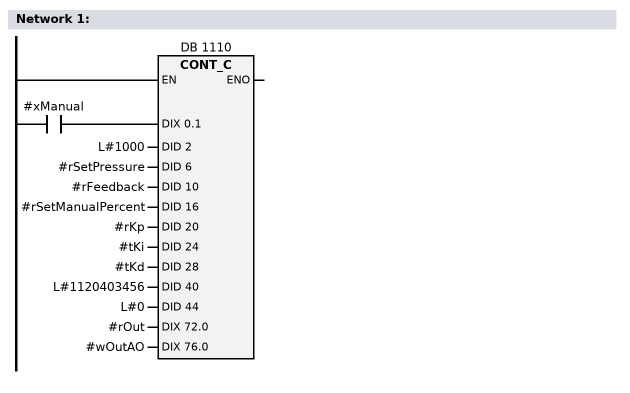
NETWORK
TITLE =
      A     #xManual;
      =     L 0.1;
      BLD   103;
      CALL  "CONT_C" , DB 1110 (
           DIX 0.1                  := L 0.1,
           DID 2                    := L#1000,
           DID 6                    := #rSetPressure,
           DID 10                   := #rFeedback,
           DID 16                   := #rSetManualPercent,
           DID 20                   := #rKp,
           DID 24                   := #tKi,
           DID 28                   := #tKd,
           DID 40                   := L#1120403456,
           DID 44                   := L#0,
           DIX 72.0                 := #rOut,
           DIX 76.0                 := #wOutAO);
      NOP   0;
END_FUNCTION_BLOCK

FUNCTION_BLOCK "fbPID"	// FB 34
VERSION : 0.1
BEGIN
// (block stored without names or comments; labels and parameter names are numbered)
END_FUNCTION_BLOCK

// FB 35: know-how protected block, not included

FUNCTION_BLOCK "DERIVATIVE"	// FB 36
VERSION : 0.0
VAR_INPUT
  IN : REAL ;
  TM : INT ;
  RESET : BOOL ;
END_VAR
VAR_OUTPUT
  OUT : REAL ;
END_VAR
VAR
  X3 : REAL ;
  X2 : REAL ;
  X1 : REAL ;
  T_2 : INT ;
  T_1 : INT ;
  INIT : BOOL  := TRUE;
END_VAR
BEGIN
// body was compiled from an SCL source; compiled code not shown
END_FUNCTION_BLOCK

FUNCTION_BLOCK "INTEGRAL"	// FB 37
VERSION : 0.0
VAR_INPUT
  IN : REAL ;
  TM : INT ;
  RESET : BOOL ;
END_VAR
VAR_OUTPUT
  OUT : REAL ;
  OVERFLOW : BOOL ;
END_VAR
BEGIN
// body was compiled from an SCL source; compiled code not shown
END_FUNCTION_BLOCK

FUNCTION_BLOCK "DO_Valve"	// FB 38
VERSION : 0.0
VAR_INPUT
  xCmdStop : BOOL ;
  xSnsOpn : BOOL ;
  xSnsCls : BOOL ;
  xAlm : BOOL ;
END_VAR
VAR_OUTPUT
  xDO_Opn : BOOL ;
  xDO_Cls : BOOL ;
  xDO_Stop : BOOL ;
END_VAR
VAR_IN_OUT
  xCmdOpn : BOOL ;
  xCmdCls : BOOL ;
END_VAR
VAR
  rtOn : BOOL ;
  rtOff : BOOL ;
  ftOn : BOOL ;
  ftOff : BOOL ;
  OpnOld : BOOL ;
  ClsOld : BOOL ;
END_VAR
BEGIN
// body was compiled from an SCL source; compiled code not shown
END_FUNCTION_BLOCK

FUNCTION_BLOCK "ValvesPrg"	// FB 39
VERSION : 0.1
BEGIN
NETWORK
TITLE =
NETWORK
TITLE =
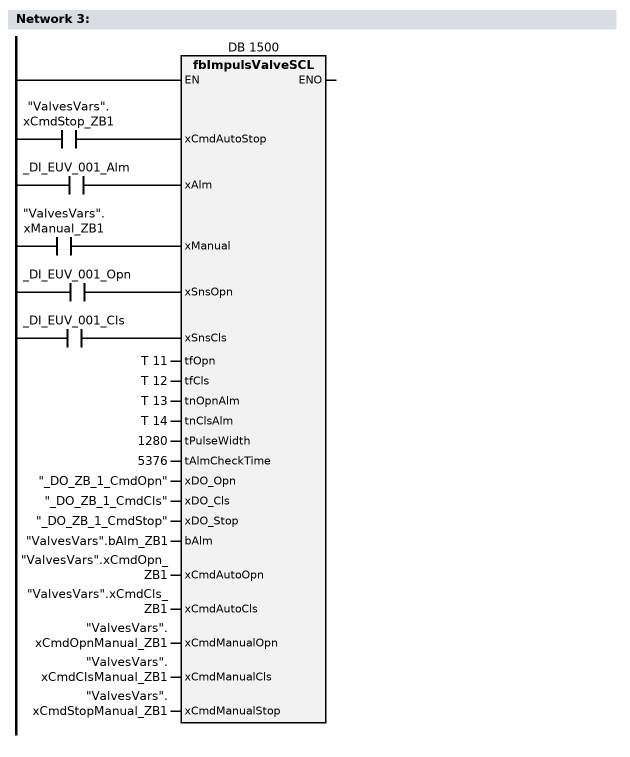
NETWORK
TITLE =
      A     "ValvesVars".xCmdStop_ZB1;
      =     L 0.0;
      BLD   103;
      A     "_DI_EUV_001_Alm";
      =     L 0.1;
      BLD   103;
      A     "ValvesVars".xManual_ZB1;
      =     L 0.2;
      BLD   103;
      A     "_DI_EUV_001_Opn";
      =     L 0.3;
      BLD   103;
      A     "_DI_EUV_001_Cls";
      =     L 0.4;
      BLD   103;
      CALL  "fbImpulsValveSCL" , DB 1500 (
           xCmdAutoStop             := L 0.0,
           xAlm                     := L 0.1,
           xManual                  := L 0.2,
           xSnsOpn                  := L 0.3,
           xSnsCls                  := L 0.4,
           tfOpn                    := T 11,
           tfCls                    := T 12,
           tnOpnAlm                 := T 13,
           tnClsAlm                 := T 14,
           tPulseWidth              := 1280,
           tAlmCheckTime            := 5376,
           xDO_Opn                  := "_DO_ZB_1_CmdOpn",
           xDO_Cls                  := "_DO_ZB_1_CmdCls",
           xDO_Stop                 := "_DO_ZB_1_CmdStop",
           bAlm                     := "ValvesVars".bAlm_ZB1,
           xCmdAutoOpn              := "ValvesVars".xCmdOpn_ZB1,
           xCmdAutoCls              := "ValvesVars".xCmdCls_ZB1,
           xCmdManualOpn            := "ValvesVars".xCmdOpnManual_ZB1,
           xCmdManualCls            := "ValvesVars".xCmdClsManual_ZB1,
           xCmdManualStop           := "ValvesVars".xCmdStopManual_ZB1);
      NOP   0;
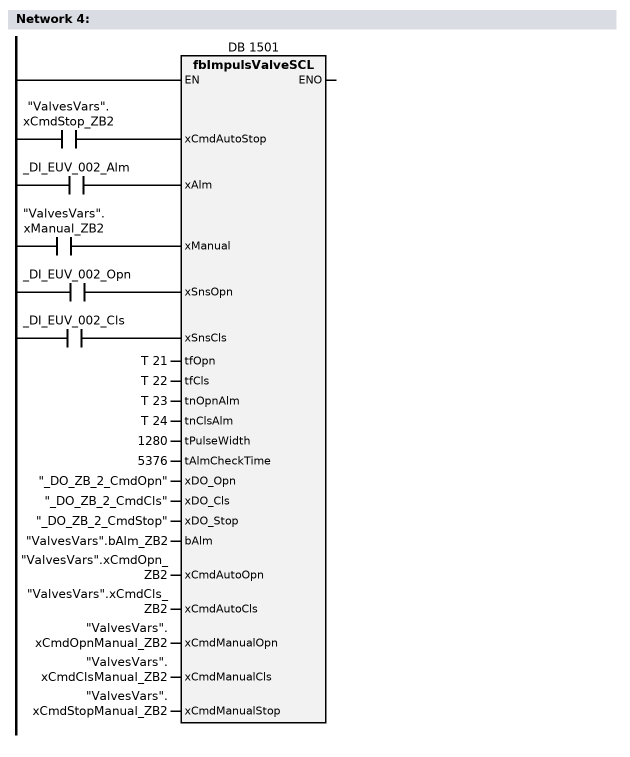
NETWORK
TITLE =
      A     "ValvesVars".xCmdStop_ZB2;
      =     L 0.0;
      BLD   103;
      A     "_DI_EUV_002_Alm";
      =     L 0.1;
      BLD   103;
      A     "ValvesVars".xManual_ZB2;
      =     L 0.2;
      BLD   103;
      A     "_DI_EUV_002_Opn";
      =     L 0.3;
      BLD   103;
      A     "_DI_EUV_002_Cls";
      =     L 0.4;
      BLD   103;
      CALL  "fbImpulsValveSCL" , DB 1501 (
           xCmdAutoStop             := L 0.0,
           xAlm                     := L 0.1,
           xManual                  := L 0.2,
           xSnsOpn                  := L 0.3,
           xSnsCls                  := L 0.4,
           tfOpn                    := T 21,
           tfCls                    := T 22,
           tnOpnAlm                 := T 23,
           tnClsAlm                 := T 24,
           tPulseWidth              := 1280,
           tAlmCheckTime            := 5376,
           xDO_Opn                  := "_DO_ZB_2_CmdOpn",
           xDO_Cls                  := "_DO_ZB_2_CmdCls",
           xDO_Stop                 := "_DO_ZB_2_CmdStop",
           bAlm                     := "ValvesVars".bAlm_ZB2,
           xCmdAutoOpn              := "ValvesVars".xCmdOpn_ZB2,
           xCmdAutoCls              := "ValvesVars".xCmdCls_ZB2,
           xCmdManualOpn            := "ValvesVars".xCmdOpnManual_ZB2,
           xCmdManualCls            := "ValvesVars".xCmdClsManual_ZB2,
           xCmdManualStop           := "ValvesVars".xCmdStopManual_ZB2);
      NOP   0;
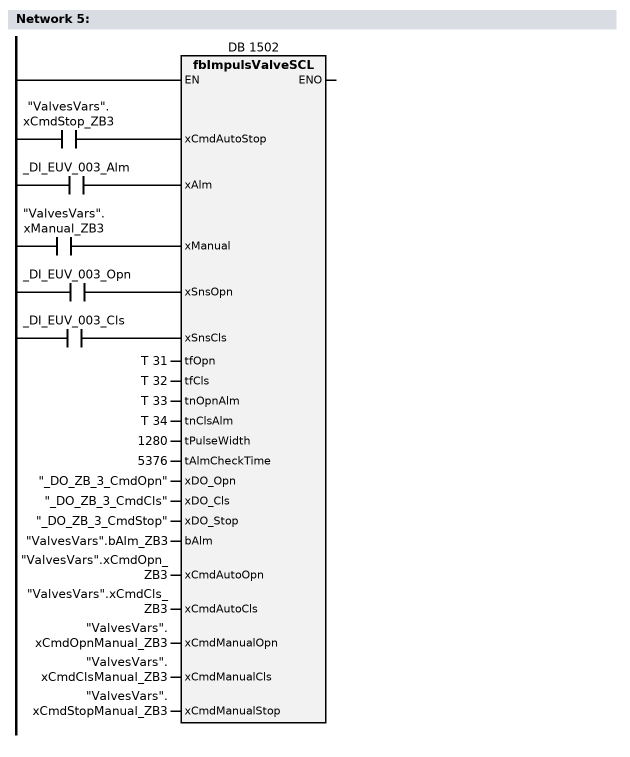
NETWORK
TITLE =
      A     "ValvesVars".xCmdStop_ZB3;
      =     L 0.0;
      BLD   103;
      A     "_DI_EUV_003_Alm";
      =     L 0.1;
      BLD   103;
      A     "ValvesVars".xManual_ZB3;
      =     L 0.2;
      BLD   103;
      A     "_DI_EUV_003_Opn";
      =     L 0.3;
      BLD   103;
      A     "_DI_EUV_003_Cls";
      =     L 0.4;
      BLD   103;
      CALL  "fbImpulsValveSCL" , DB 1502 (
           xCmdAutoStop             := L 0.0,
           xAlm                     := L 0.1,
           xManual                  := L 0.2,
           xSnsOpn                  := L 0.3,
           xSnsCls                  := L 0.4,
           tfOpn                    := T 31,
           tfCls                    := T 32,
           tnOpnAlm                 := T 33,
           tnClsAlm                 := T 34,
           tPulseWidth              := 1280,
           tAlmCheckTime            := 5376,
           xDO_Opn                  := "_DO_ZB_3_CmdOpn",
           xDO_Cls                  := "_DO_ZB_3_CmdCls",
           xDO_Stop                 := "_DO_ZB_3_CmdStop",
           bAlm                     := "ValvesVars".bAlm_ZB3,
           xCmdAutoOpn              := "ValvesVars".xCmdOpn_ZB3,
           xCmdAutoCls              := "ValvesVars".xCmdCls_ZB3,
           xCmdManualOpn            := "ValvesVars".xCmdOpnManual_ZB3,
           xCmdManualCls            := "ValvesVars".xCmdClsManual_ZB3,
           xCmdManualStop           := "ValvesVars".xCmdStopManual_ZB3);
      NOP   0;
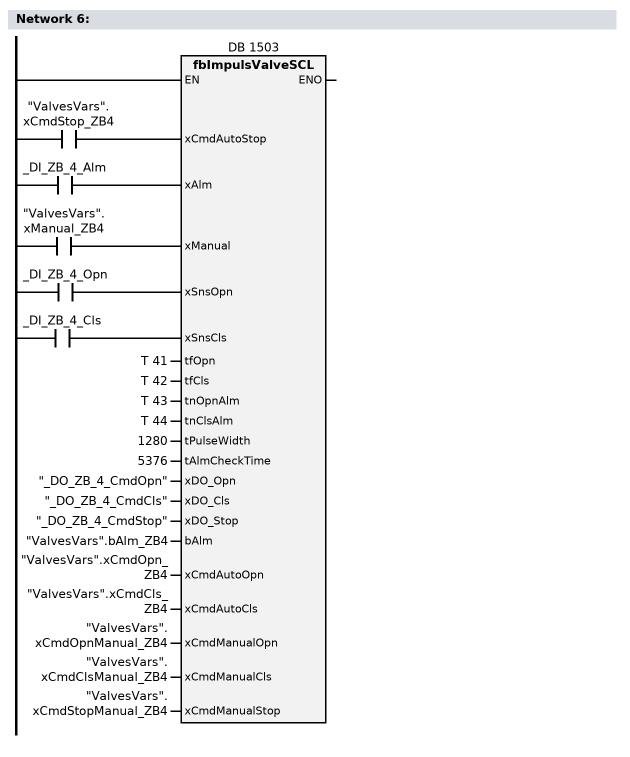
NETWORK
TITLE =
      A     "ValvesVars".xCmdStop_ZB4;
      =     L 0.0;
      BLD   103;
      A     "_DI_ZB_4_Alm";
      =     L 0.1;
      BLD   103;
      A     "ValvesVars".xManual_ZB4;
      =     L 0.2;
      BLD   103;
      A     "_DI_ZB_4_Opn";
      =     L 0.3;
      BLD   103;
      A     "_DI_ZB_4_Cls";
      =     L 0.4;
      BLD   103;
      CALL  "fbImpulsValveSCL" , DB 1503 (
           xCmdAutoStop             := L 0.0,
           xAlm                     := L 0.1,
           xManual                  := L 0.2,
           xSnsOpn                  := L 0.3,
           xSnsCls                  := L 0.4,
           tfOpn                    := T 41,
           tfCls                    := T 42,
           tnOpnAlm                 := T 43,
           tnClsAlm                 := T 44,
           tPulseWidth              := 1280,
           tAlmCheckTime            := 5376,
           xDO_Opn                  := "_DO_ZB_4_CmdOpn",
           xDO_Cls                  := "_DO_ZB_4_CmdCls",
           xDO_Stop                 := "_DO_ZB_4_CmdStop",
           bAlm                     := "ValvesVars".bAlm_ZB4,
           xCmdAutoOpn              := "ValvesVars".xCmdOpn_ZB4,
           xCmdAutoCls              := "ValvesVars".xCmdCls_ZB4,
           xCmdManualOpn            := "ValvesVars".xCmdOpnManual_ZB4,
           xCmdManualCls            := "ValvesVars".xCmdClsManual_ZB4,
           xCmdManualStop           := "ValvesVars".xCmdStopManual_ZB4);
      NOP   0;
NETWORK
TITLE =
NETWORK
TITLE =
NETWORK
TITLE =
END_FUNCTION_BLOCK

FUNCTION_BLOCK "fbProcess_1"	// FB 40
VERSION : 0.0
VAR_INPUT
  xPO_1_On : BOOL ;
  xPO_2_On : BOOL ;
  xKB1_On : BOOL ;
  xKB2_On : BOOL ;
  xKZA1_On : BOOL ;
  xKZA2_On : BOOL ;
  rPressure_PB1 : REAL ;
  rPressure_PB2 : REAL ;
  rPressure_Set : REAL ;
  xTM_KB1_Q : BOOL ;
  xTM_KB2_Q : BOOL ;
END_VAR
VAR_OUTPUT
  wState : INT ;
  xStartTM_KB1 : BOOL ;
  xStartTM_KB2 : BOOL ;
END_VAR
VAR_IN_OUT
  xStart : BOOL ;
  xPO_1_CmdStart : BOOL ;
  xPO_2_CmdStart : BOOL ;
  xKB1_CmdStart : BOOL ;
  xKB2_CmdStart : BOOL ;
  xKZA1_CmdStart : BOOL ;
  xKZA2_CmdStart : BOOL ;
  xPO_1_CmdStop : BOOL ;
  xPO_2_CmdStop : BOOL ;
  xKB1_CmdStop : BOOL ;
  xKB2_CmdStop : BOOL ;
  xKZA1_CmdStop : BOOL ;
  xKZA2_CmdStop : BOOL ;
END_VAR
BEGIN
// body was compiled from an SCL source; compiled code not shown
END_FUNCTION_BLOCK

// FB 41: know-how protected block, not included

// FB 42: know-how protected block, not included

FUNCTION_BLOCK "fbImpulsValve"	// FB 43
VERSION : 0.1
VAR_INPUT
  xOpn : BOOL ;
  xCls : BOOL ;
  xStop : BOOL ;
END_VAR
VAR_OUTPUT
  xDO_Opn : BOOL ;
  xDO_Cls : BOOL ;
  xDO_Stop : BOOL ;
END_VAR
VAR_TEMP
  xOpen : BOOL ;
  xClose : BOOL ;
END_VAR
BEGIN
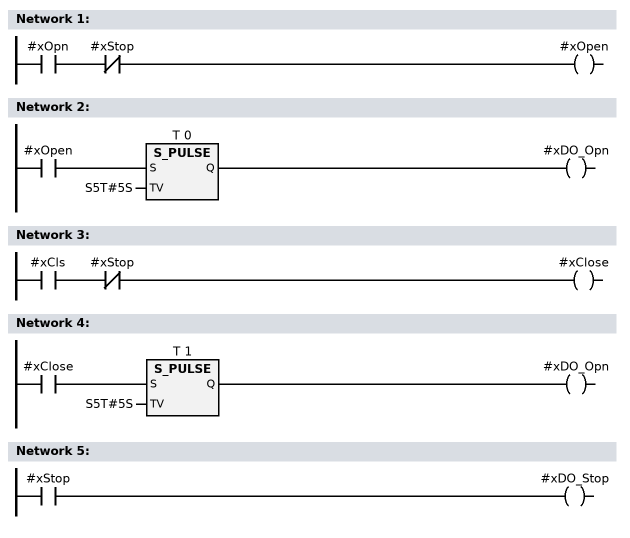
NETWORK
TITLE =
      A     #xOpn;
      AN    #xStop;
      =     #xOpen;
NETWORK
TITLE =
      A     #xOpen;
      L     S5T#5S;
      SP    T 0;
      NOP   0;
      NOP   0;
      NOP   0;
      A     T 0;
      =     #xDO_Opn;
NETWORK
TITLE =
      A     #xCls;
      AN    #xStop;
      =     #xClose;
NETWORK
TITLE =
      A     #xClose;
      L     S5T#5S;
      SP    T 1;
      NOP   0;
      NOP   0;
      NOP   0;
      A     T 1;
      =     #xDO_Opn;
NETWORK
TITLE =
      A     #xStop;
      =     #xDO_Stop;
END_FUNCTION_BLOCK

FUNCTION_BLOCK "fbImpulsValveSCL"	// FB 44
VERSION : 0.0
VAR_INPUT
  xCmdAutoStop : BOOL ;
  xAlm : BOOL ;
  xManual : BOOL ;
  xSnsOpn : BOOL ;
  xSnsCls : BOOL ;
  tfOpn : TIMER ;
  tfCls : TIMER ;
  tnOpnAlm : TIMER ;
  tnClsAlm : TIMER ;
  tPulseWidth : S5TIME ;
  tAlmCheckTime : S5TIME ;
END_VAR
VAR_OUTPUT
  xDO_Opn : BOOL ;
  xDO_Cls : BOOL ;
  xDO_Stop : BOOL ;
  bAlm : BYTE ;
END_VAR
VAR_IN_OUT
  xCmdAutoOpn : BOOL ;
  xCmdAutoCls : BOOL ;
  xCmdManualOpn : BOOL ;
  xCmdManualCls : BOOL ;
  xCmdManualStop : BOOL ;
  xResetAlm : BOOL ;
END_VAR
VAR
  xManualOld : BOOL ;
  currTime : S5TIME ;
  currTime1 : S5TIME ;
  currTime2 : S5TIME ;
  currTime13 : S5TIME ;
  xAlmOpnTON_Q : BOOL ;
  xAlmOpnTON_Q_Old : BOOL ;
  xAlmClsTON_Q : BOOL ;
  xAlmClsTON_Q_Old : BOOL ;
END_VAR
BEGIN
// body was compiled from an SCL source; compiled code not shown
END_FUNCTION_BLOCK

FUNCTION_BLOCK "prProcess"	// FB 45
VERSION : 0.1
VAR_TEMP
  xStartTON_1 : BOOL ;
  xStartTON_2 : BOOL ;
  xTON_1_Q : BOOL ;
  xTON_2_Q : BOOL ;
  xTON_1_Q_1 : BOOL ;
  xTON_2_Q_1 : BOOL ;
  xPlug : BOOL ;
  xStartTON_1_1 : BOOL ;
  xStartTON_2_1 : BOOL ;
END_VAR
BEGIN
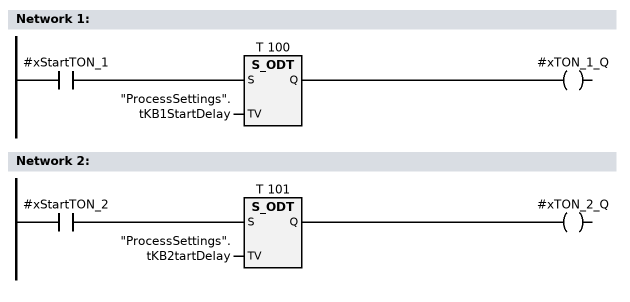
NETWORK
TITLE =
      A     #xStartTON_1;
      L     "ProcessSettings".tKB1StartDelay;
      SD    T 100;
      NOP   0;
      NOP   0;
      NOP   0;
      A     T 100;
      =     #xTON_1_Q;
NETWORK
TITLE =
      A     #xStartTON_2;
      L     "ProcessSettings".tKB2tartDelay;
      SD    T 101;
      NOP   0;
      NOP   0;
      NOP   0;
      A     T 101;
      =     #xTON_2_Q;
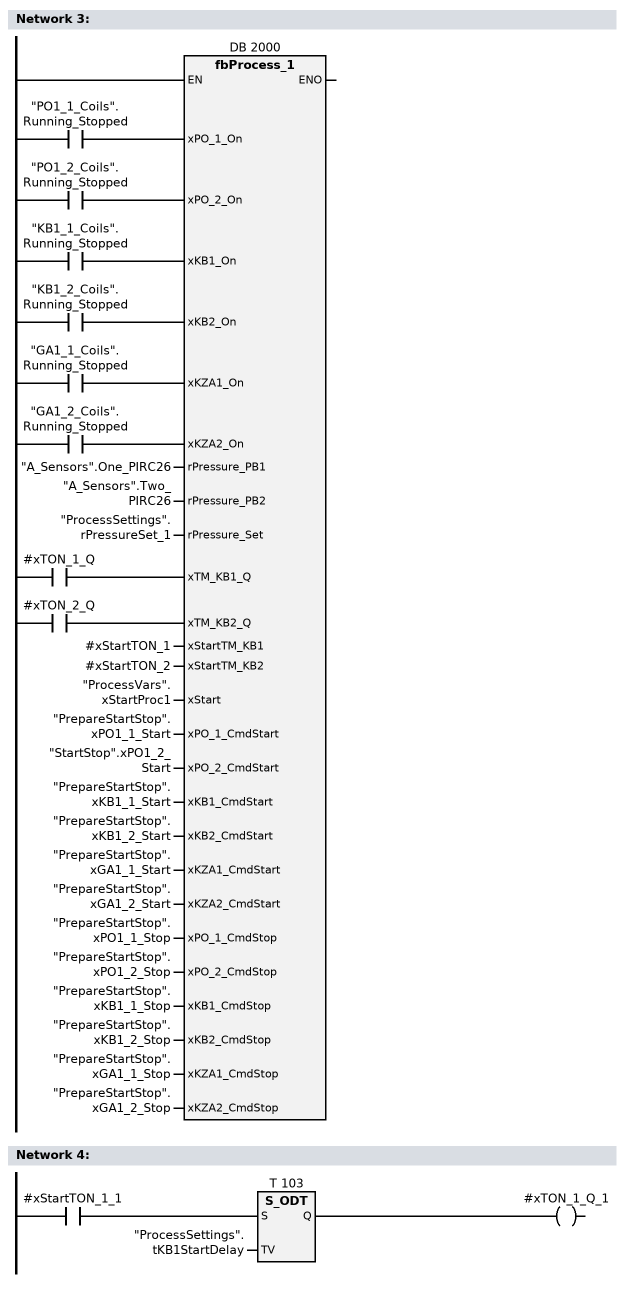
NETWORK
TITLE =
      A     "PO1_1_Coils".Running_Stopped;
      =     L 2.0;
      BLD   103;
      A     "PO1_2_Coils".Running_Stopped;
      =     L 2.1;
      BLD   103;
      A     "KB1_1_Coils".Running_Stopped;
      =     L 2.2;
      BLD   103;
      A     "KB1_2_Coils".Running_Stopped;
      =     L 2.3;
      BLD   103;
      A     "GA1_1_Coils".Running_Stopped;
      =     L 2.4;
      BLD   103;
      A     "GA1_2_Coils".Running_Stopped;
      =     L 2.5;
      BLD   103;
      A     #xTON_1_Q;
      =     L 2.6;
      BLD   103;
      A     #xTON_2_Q;
      =     L 2.7;
      BLD   103;
      CALL  "fbProcess_1" , DB 2000 (
           xPO_1_On                 := L 2.0,
           xPO_2_On                 := L 2.1,
           xKB1_On                  := L 2.2,
           xKB2_On                  := L 2.3,
           xKZA1_On                 := L 2.4,
           xKZA2_On                 := L 2.5,
           rPressure_PB1            := "A_Sensors".One_PIRC26,
           rPressure_PB2            := "A_Sensors".Two_PIRC26,
           rPressure_Set            := "ProcessSettings".rPressureSet_1,
           xTM_KB1_Q                := L 2.6,
           xTM_KB2_Q                := L 2.7,
           xStartTM_KB1             := #xStartTON_1,
           xStartTM_KB2             := #xStartTON_2,
           xStart                   := "ProcessVars".xStartProc1,
           xPO_1_CmdStart           := "PrepareStartStop".xPO1_1_Start,
           xPO_2_CmdStart           := "StartStop".xPO1_2_Start,
           xKB1_CmdStart            := "PrepareStartStop".xKB1_1_Start,
           xKB2_CmdStart            := "PrepareStartStop".xKB1_2_Start,
           xKZA1_CmdStart           := "PrepareStartStop".xGA1_1_Start,
           xKZA2_CmdStart           := "PrepareStartStop".xGA1_2_Start,
           xPO_1_CmdStop            := "PrepareStartStop".xPO1_1_Stop,
           xPO_2_CmdStop            := "PrepareStartStop".xPO1_2_Stop,
           xKB1_CmdStop             := "PrepareStartStop".xKB1_1_Stop,
           xKB2_CmdStop             := "PrepareStartStop".xKB1_2_Stop,
           xKZA1_CmdStop            := "PrepareStartStop".xGA1_1_Stop,
           xKZA2_CmdStop            := "PrepareStartStop".xGA1_2_Stop);
      NOP   0;
NETWORK
TITLE =
      A     #xStartTON_1_1;
      L     "ProcessSettings".tKB1StartDelay;
      SD    T 103;
      NOP   0;
      NOP   0;
      NOP   0;
      A     T 103;
      =     #xTON_1_Q_1;
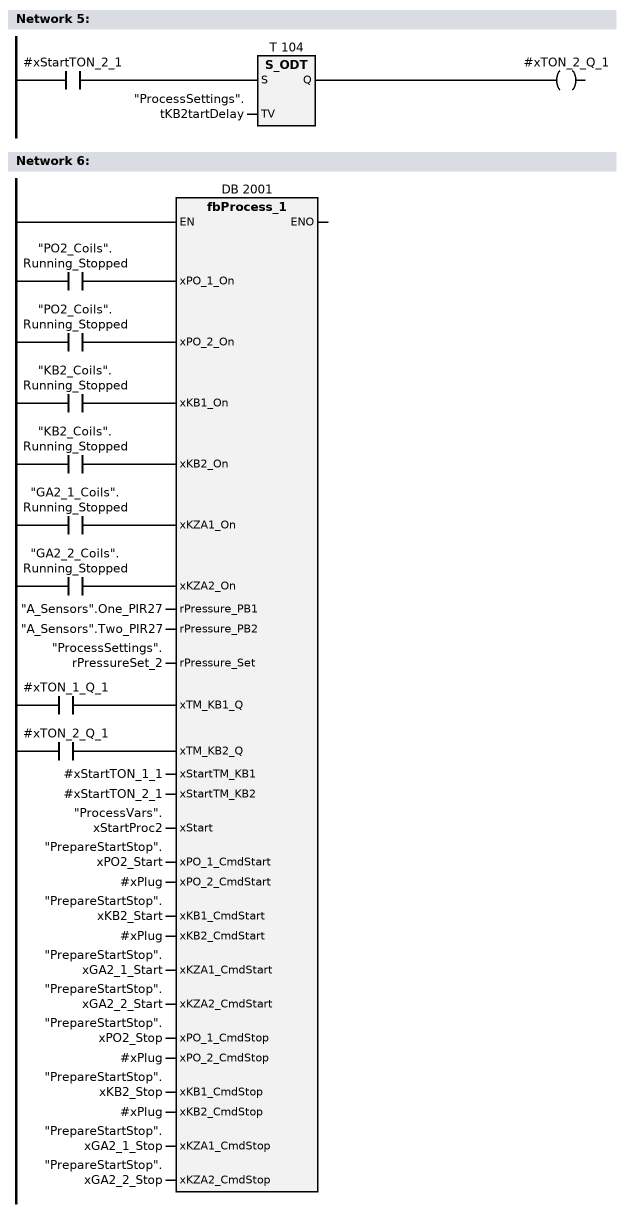
NETWORK
TITLE =
      A     #xStartTON_2_1;
      L     "ProcessSettings".tKB2tartDelay;
      SD    T 104;
      NOP   0;
      NOP   0;
      NOP   0;
      A     T 104;
      =     #xTON_2_Q_1;
NETWORK
TITLE =
      A     "PO2_Coils".Running_Stopped;
      =     L 2.0;
      BLD   103;
      A     "PO2_Coils".Running_Stopped;
      =     L 2.1;
      BLD   103;
      A     "KB2_Coils".Running_Stopped;
      =     L 2.2;
      BLD   103;
      A     "KB2_Coils".Running_Stopped;
      =     L 2.3;
      BLD   103;
      A     "GA2_1_Coils".Running_Stopped;
      =     L 2.4;
      BLD   103;
      A     "GA2_2_Coils".Running_Stopped;
      =     L 2.5;
      BLD   103;
      A     #xTON_1_Q_1;
      =     L 2.6;
      BLD   103;
      A     #xTON_2_Q_1;
      =     L 2.7;
      BLD   103;
      CALL  "fbProcess_1" , DB 2001 (
           xPO_1_On                 := L 2.0,
           xPO_2_On                 := L 2.1,
           xKB1_On                  := L 2.2,
           xKB2_On                  := L 2.3,
           xKZA1_On                 := L 2.4,
           xKZA2_On                 := L 2.5,
           rPressure_PB1            := "A_Sensors".One_PIR27,
           rPressure_PB2            := "A_Sensors".Two_PIR27,
           rPressure_Set            := "ProcessSettings".rPressureSet_2,
           xTM_KB1_Q                := L 2.6,
           xTM_KB2_Q                := L 2.7,
           xStartTM_KB1             := #xStartTON_1_1,
           xStartTM_KB2             := #xStartTON_2_1,
           xStart                   := "ProcessVars".xStartProc2,
           xPO_1_CmdStart           := "PrepareStartStop".xPO2_Start,
           xPO_2_CmdStart           := #xPlug,
           xKB1_CmdStart            := "PrepareStartStop".xKB2_Start,
           xKB2_CmdStart            := #xPlug,
           xKZA1_CmdStart           := "PrepareStartStop".xGA2_1_Start,
           xKZA2_CmdStart           := "PrepareStartStop".xGA2_2_Start,
           xPO_1_CmdStop            := "PrepareStartStop".xPO2_Stop,
           xPO_2_CmdStop            := #xPlug,
           xKB1_CmdStop             := "PrepareStartStop".xKB2_Stop,
           xKB2_CmdStop             := #xPlug,
           xKZA1_CmdStop            := "PrepareStartStop".xGA2_1_Stop,
           xKZA2_CmdStop            := "PrepareStartStop".xGA2_2_Stop);
      NOP   0;
END_FUNCTION_BLOCK

FUNCTION_BLOCK "fbPO"	// FB 46
VERSION : 0.0
VAR_INPUT
  xPO_Working : BOOL ;
  tnWotkingTimer : TIMER ;
  tSetWorkingTime : S5TIME ;
END_VAR
VAR_OUTPUT
  xTimeElapsed : BOOL ;
END_VAR
VAR
  currTime : S5TIME ;
END_VAR
BEGIN
// body was compiled from an SCL source; compiled code not shown
END_FUNCTION_BLOCK

FUNCTION_BLOCK "fbKB"	// FB 47
VERSION : 0.0
VAR_INPUT
  xInterlock : BOOL ;
END_VAR
VAR_OUTPUT
  xOutStart : BOOL ;
  xOutStop : BOOL ;
END_VAR
VAR_IN_OUT
  xStart : BOOL ;
  xStop : BOOL ;
END_VAR
VAR
  currTime : S5TIME ;
END_VAR
BEGIN
// body was compiled from an SCL source; compiled code not shown
END_FUNCTION_BLOCK

FUNCTION_BLOCK "fbKZA"	// FB 48
VERSION : 0.0
VAR_INPUT
  rPressureSet : REAL ;
  rPressureGet : REAL ;
  rHyster : REAL  := 2.000000e-001;
END_VAR
VAR_OUTPUT
  xOutStart : BOOL ;
  xOutStop : BOOL ;
END_VAR
VAR_IN_OUT
  xStart : BOOL ;
  xStop : BOOL ;
END_VAR
BEGIN
// body was compiled from an SCL source; compiled code not shown
END_FUNCTION_BLOCK

FUNCTION_BLOCK "prDevices"	// FB 49
VERSION : 0.1
VAR_TEMP
  xKB1_1_Interlock : BOOL ;
  xKB1_2_Interlock : BOOL ;
  xKB2_Interlock : BOOL ;
END_VAR
BEGIN
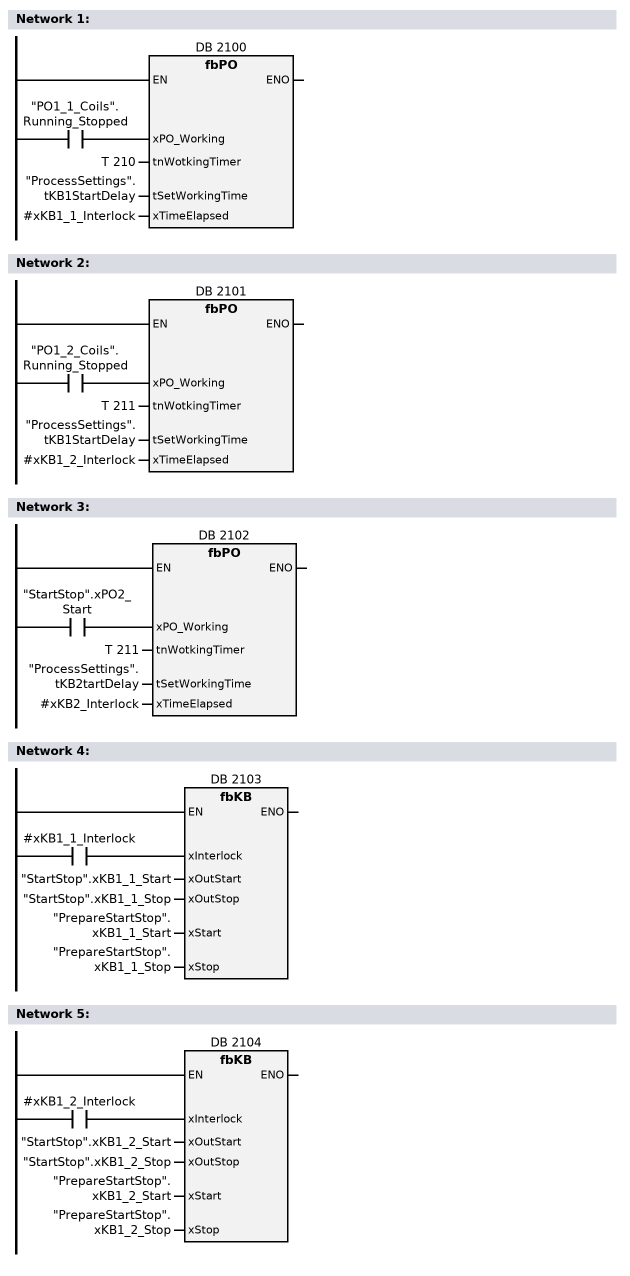
NETWORK
TITLE =
      A     "PO1_1_Coils".Running_Stopped;
      =     L 1.0;
      BLD   103;
      CALL  "fbPO" , DB 2100 (
           xPO_Working              := L 1.0,
           tnWotkingTimer           := T 210,
           tSetWorkingTime          := "ProcessSettings".tKB1StartDelay,
           xTimeElapsed             := #xKB1_1_Interlock);
      NOP   0;
NETWORK
TITLE =
      A     "PO1_2_Coils".Running_Stopped;
      =     L 1.0;
      BLD   103;
      CALL  "fbPO" , DB 2101 (
           xPO_Working              := L 1.0,
           tnWotkingTimer           := T 211,
           tSetWorkingTime          := "ProcessSettings".tKB1StartDelay,
           xTimeElapsed             := #xKB1_2_Interlock);
      NOP   0;
NETWORK
TITLE =
      A     "StartStop".xPO2_Start;
      =     L 1.0;
      BLD   103;
      CALL  "fbPO" , DB 2102 (
           xPO_Working              := L 1.0,
           tnWotkingTimer           := T 211,
           tSetWorkingTime          := "ProcessSettings".tKB2tartDelay,
           xTimeElapsed             := #xKB2_Interlock);
      NOP   0;
NETWORK
TITLE =
      A     #xKB1_1_Interlock;
      =     L 1.0;
      BLD   103;
      CALL  "fbKB" , DB 2103 (
           xInterlock               := L 1.0,
           xOutStart                := "StartStop".xKB1_1_Start,
           xOutStop                 := "StartStop".xKB1_1_Stop,
           xStart                   := "PrepareStartStop".xKB1_1_Start,
           xStop                    := "PrepareStartStop".xKB1_1_Stop);
      NOP   0;
NETWORK
TITLE =
      A     #xKB1_2_Interlock;
      =     L 1.0;
      BLD   103;
      CALL  "fbKB" , DB 2104 (
           xInterlock               := L 1.0,
           xOutStart                := "StartStop".xKB1_2_Start,
           xOutStop                 := "StartStop".xKB1_2_Stop,
           xStart                   := "PrepareStartStop".xKB1_2_Start,
           xStop                    := "PrepareStartStop".xKB1_2_Stop);
      NOP   0;
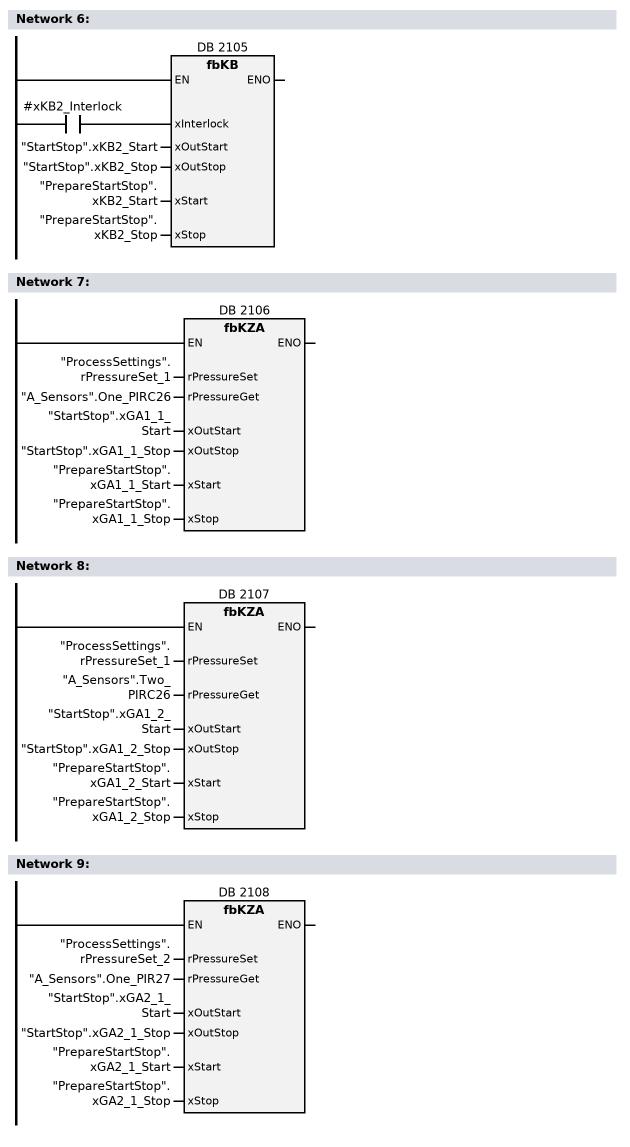
NETWORK
TITLE =
      A     #xKB2_Interlock;
      =     L 1.0;
      BLD   103;
      CALL  "fbKB" , DB 2105 (
           xInterlock               := L 1.0,
           xOutStart                := "StartStop".xKB2_Start,
           xOutStop                 := "StartStop".xKB2_Stop,
           xStart                   := "PrepareStartStop".xKB2_Start,
           xStop                    := "PrepareStartStop".xKB2_Stop);
      NOP   0;
NETWORK
TITLE =
      CALL  "fbKZA" , DB 2106 (
           rPressureSet             := "ProcessSettings".rPressureSet_1,
           rPressureGet             := "A_Sensors".One_PIRC26,
           xOutStart                := "StartStop".xGA1_1_Start,
           xOutStop                 := "StartStop".xGA1_1_Stop,
           xStart                   := "PrepareStartStop".xGA1_1_Start,
           xStop                    := "PrepareStartStop".xGA1_1_Stop);
      NOP   0;
NETWORK
TITLE =
      CALL  "fbKZA" , DB 2107 (
           rPressureSet             := "ProcessSettings".rPressureSet_1,
           rPressureGet             := "A_Sensors".Two_PIRC26,
           xOutStart                := "StartStop".xGA1_2_Start,
           xOutStop                 := "StartStop".xGA1_2_Stop,
           xStart                   := "PrepareStartStop".xGA1_2_Start,
           xStop                    := "PrepareStartStop".xGA1_2_Stop);
      NOP   0;
NETWORK
TITLE =
      CALL  "fbKZA" , DB 2108 (
           rPressureSet             := "ProcessSettings".rPressureSet_2,
           rPressureGet             := "A_Sensors".One_PIR27,
           xOutStart                := "StartStop".xGA2_1_Start,
           xOutStop                 := "StartStop".xGA2_1_Stop,
           xStart                   := "PrepareStartStop".xGA2_1_Start,
           xStop                    := "PrepareStartStop".xGA2_1_Stop);
      NOP   0;
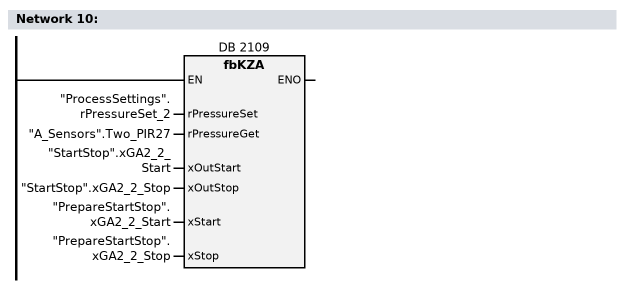
NETWORK
TITLE =
      CALL  "fbKZA" , DB 2109 (
           rPressureSet             := "ProcessSettings".rPressureSet_2,
           rPressureGet             := "A_Sensors".Two_PIR27,
           xOutStart                := "StartStop".xGA2_2_Start,
           xOutStop                 := "StartStop".xGA2_2_Stop,
           xStart                   := "PrepareStartStop".xGA2_2_Start,
           xStop                    := "PrepareStartStop".xGA2_2_Stop);
      NOP   0;
END_FUNCTION_BLOCK

FUNCTION_BLOCK "GetCoils"	// FB 50
VERSION : 0.1
BEGIN
NETWORK
TITLE =
      A     "BD_Coils".Running_Stopped;
      =     DB6.DBX 0.0;
      A     "BD_Coils".Load_Unload;
      =     DB6.DBX 0.1;
      A     "BD_Coils".General_Warning;
      =     DB6.DBX 0.2;
      A     "BD_Coils".GeneralShutdownWarning;
      =     DB6.DBX 0.3;
      A     "BD_Coils".GeneralShutdown;
      =     DB6.DBX 0.4;
      A     "BD_Coils".GeneralService;
      =     DB6.DBX 0.5;
      A     "BD_Coils".GeneralStartFailure;
      =     DB6.DBX 0.6;
      A     "BD_Coils".EmergencyStop;
      =     DB6.DBX 0.7;
      A     "BD_Coils".Automatic_Manual;
      =     DB6.DBX 1.0;
      A     "BD_Coils".Remote_Local;
      =     DB6.DBX 1.1;
      A     "GA1_1_Coils".Running_Stopped;
      =     DB12.DBX 0.0;
      A     "GA1_1_Coils".Load_Unload;
      =     DB12.DBX 0.1;
      A     "GA1_1_Coils".General_Warning;
      =     DB12.DBX 0.2;
      A     "GA1_1_Coils".GeneralShutdownWarning;
      =     DB12.DBX 0.3;
      A     "GA1_1_Coils".GeneralShutdown;
      =     DB12.DBX 0.4;
      A     "GA1_1_Coils".GeneralService;
      =     DB12.DBX 0.5;
      A     "GA1_1_Coils".GeneralStartFailure;
      =     DB12.DBX 0.6;
      A     "GA1_1_Coils".EmergencyStop;
      =     DB12.DBX 0.7;
      A     "GA1_1_Coils".Automatic_Manual;
      =     DB12.DBX 1.0;
      A     "GA1_1_Coils".Remote_Local;
      =     DB12.DBX 1.1;
      A     "GA1_2_Coils".Running_Stopped;
      =     DB13.DBX 0.0;
      A     "GA1_2_Coils".Load_Unload;
      =     DB13.DBX 0.1;
      A     "GA1_2_Coils".General_Warning;
      =     DB13.DBX 0.2;
      A     "GA1_2_Coils".GeneralShutdownWarning;
      =     DB13.DBX 0.3;
      A     "GA1_2_Coils".GeneralShutdown;
      =     DB13.DBX 0.4;
      A     "GA1_2_Coils".GeneralService;
      =     DB13.DBX 0.5;
      A     "GA1_2_Coils".GeneralStartFailure;
      =     DB13.DBX 0.6;
      A     "GA1_2_Coils".EmergencyStop;
      =     DB13.DBX 0.7;
      A     "GA1_2_Coils".Automatic_Manual;
      =     DB13.DBX 1.0;
      A     "GA1_2_Coils".Remote_Local;
      =     DB13.DBX 1.1;
      A     "GA2_1_Coils".Running_Stopped;
      =     DB14.DBX 0.0;
      A     "GA2_1_Coils".Load_Unload;
      =     DB14.DBX 0.1;
      A     "GA2_1_Coils".General_Warning;
      =     DB14.DBX 0.2;
      A     "GA2_1_Coils".GeneralShutdownWarning;
      =     DB14.DBX 0.3;
      A     "GA2_1_Coils".GeneralShutdown;
      =     DB14.DBX 0.4;
      A     "GA2_1_Coils".GeneralService;
      =     DB14.DBX 0.5;
      A     "GA2_1_Coils".GeneralStartFailure;
      =     DB14.DBX 0.6;
      A     "GA2_1_Coils".EmergencyStop;
      =     DB14.DBX 0.7;
      A     "GA2_1_Coils".Automatic_Manual;
      =     DB14.DBX 1.0;
      A     "GA2_1_Coils".Remote_Local;
      =     DB14.DBX 1.1;
      A     "GA2_2_Coils".Running_Stopped;
      =     DB15.DBX 0.0;
      A     "GA2_2_Coils".Load_Unload;
      =     DB15.DBX 0.1;
      A     "GA2_2_Coils".General_Warning;
      =     DB15.DBX 0.2;
      A     "GA2_2_Coils".GeneralShutdownWarning;
      =     DB15.DBX 0.3;
      A     "GA2_2_Coils".GeneralShutdown;
      =     DB15.DBX 0.4;
      A     "GA2_2_Coils".GeneralService;
      =     DB15.DBX 0.5;
      A     "GA2_2_Coils".GeneralStartFailure;
      =     DB15.DBX 0.6;
      A     "GA2_2_Coils".EmergencyStop;
      =     DB15.DBX 0.7;
      A     "GA2_2_Coils".Automatic_Manual;
      =     DB15.DBX 1.0;
      A     "GA2_2_Coils".Remote_Local;
      =     DB15.DBX 1.1;
      A     "KB1_1_Coils".Running_Stopped;
      =     DB7.DBX 0.0;
      A     "KB1_1_Coils".Load_Unload;
      =     DB7.DBX 0.1;
      A     "KB1_1_Coils".General_Warning;
      =     DB7.DBX 0.2;
      A     "KB1_1_Coils".GeneralShutdownWarning;
      =     DB7.DBX 0.3;
      A     "KB1_1_Coils".GeneralShutdown;
      =     DB7.DBX 0.4;
      A     "KB1_1_Coils".GeneralService;
      =     DB7.DBX 0.5;
      A     "KB1_1_Coils".GeneralStartFailure;
      =     DB7.DBX 0.6;
      A     "KB1_1_Coils".EmergencyStop;
      =     DB7.DBX 0.7;
      A     "KB1_1_Coils".Automatic_Manual;
      =     DB7.DBX 1.0;
      A     "KB1_1_Coils".Remote_Local;
      =     DB7.DBX 1.1;
      A     "KB1_2_Coils".Running_Stopped;
      =     DB8.DBX 0.0;
      A     "KB1_2_Coils".Load_Unload;
      =     DB8.DBX 0.1;
      A     "KB1_2_Coils".General_Warning;
      =     DB8.DBX 0.2;
      A     "KB1_2_Coils".GeneralShutdownWarning;
      =     DB8.DBX 0.3;
      A     "KB1_2_Coils".GeneralShutdown;
      =     DB8.DBX 0.4;
      A     "KB1_2_Coils".GeneralService;
      =     DB8.DBX 0.5;
      A     "KB1_2_Coils".GeneralStartFailure;
      =     DB8.DBX 0.6;
      A     "KB1_2_Coils".EmergencyStop;
      =     DB8.DBX 0.7;
      A     "KB1_2_Coils".Automatic_Manual;
      =     DB8.DBX 1.0;
      A     "KB1_2_Coils".Remote_Local;
      =     DB8.DBX 1.1;
      A     "KB2_Coils".Running_Stopped;
      =     DB9.DBX 0.0;
      A     "KB2_Coils".Load_Unload;
      =     DB9.DBX 0.1;
      A     "KB2_Coils".General_Warning;
      =     DB9.DBX 0.2;
      A     "KB2_Coils".GeneralShutdownWarning;
      =     DB9.DBX 0.3;
      A     "KB2_Coils".GeneralShutdown;
      =     DB9.DBX 0.4;
      A     "KB2_Coils".GeneralService;
      =     DB9.DBX 0.5;
      A     "KB2_Coils".GeneralStartFailure;
      =     DB9.DBX 0.6;
      A     "KB2_Coils".EmergencyStop;
      =     DB9.DBX 0.7;
      A     "KB2_Coils".Automatic_Manual;
      =     DB9.DBX 1.0;
      A     "KB2_Coils".Remote_Local;
      =     DB9.DBX 1.1;
      A     "PO1_1_Coils".Running_Stopped;
      =     DB10.DBX 0.0;
      A     "PO1_1_Coils".Load_Unload;
      =     DB10.DBX 0.1;
      A     "PO1_1_Coils".General_Warning;
      =     DB10.DBX 0.2;
      A     "PO1_1_Coils".GeneralShutdownWarning;
      =     DB10.DBX 0.3;
      A     "PO1_1_Coils".GeneralShutdown;
      =     DB10.DBX 0.4;
      A     "PO1_1_Coils".GeneralService;
      =     DB10.DBX 0.5;
      A     "PO1_1_Coils".GeneralStartFailure;
      =     DB10.DBX 0.6;
      A     "PO1_1_Coils".EmergencyStop;
      =     DB10.DBX 0.7;
      A     "PO1_1_Coils".Automatic_Manual;
      =     DB10.DBX 1.0;
      A     "PO1_1_Coils".Remote_Local;
      =     DB10.DBX 1.1;
      A     "PO1_2_Coils".Running_Stopped;
      =     DB11.DBX 0.0;
      A     "PO1_2_Coils".Load_Unload;
      =     DB11.DBX 0.1;
      A     "PO1_2_Coils".General_Warning;
      =     DB11.DBX 0.2;
      A     "PO1_2_Coils".GeneralShutdownWarning;
      =     DB11.DBX 0.3;
      A     "PO1_2_Coils".GeneralShutdown;
      =     DB11.DBX 0.4;
      A     "PO1_2_Coils".GeneralService;
      =     DB11.DBX 0.5;
      A     "PO1_2_Coils".GeneralStartFailure;
      =     DB11.DBX 0.6;
      A     "PO1_2_Coils".EmergencyStop;
      =     DB11.DBX 0.7;
      A     "PO1_2_Coils".Automatic_Manual;
      =     DB11.DBX 1.0;
      A     "PO1_2_Coils".Remote_Local;
      =     DB11.DBX 1.1;
      A     "PO2_Coils".Running_Stopped;
      =     DB154.DBX 0.0;
      A     "PO2_Coils".Load_Unload;
      =     DB154.DBX 0.1;
      A     "PO2_Coils".General_Warning;
      =     DB154.DBX 0.2;
      A     "PO2_Coils".GeneralShutdownWarning;
      =     DB154.DBX 0.3;
      A     "PO2_Coils".GeneralShutdown;
      =     DB154.DBX 0.4;
      A     "PO2_Coils".GeneralService;
      =     DB154.DBX 0.5;
      A     "PO2_Coils".GeneralStartFailure;
      =     DB154.DBX 0.6;
      A     "PO2_Coils".EmergencyStop;
      =     DB154.DBX 0.7;
      A     "PO2_Coils".Automatic_Manual;
      =     DB154.DBX 1.0;
      A     "PO2_Coils".Remote_Local;
      =     DB154.DBX 1.1;
END_FUNCTION_BLOCK

FUNCTION "LinTrafo" : VOID	// FC 1
VERSION : 0.0
VAR_INPUT
  IN_WORD : WORD ;
  IN_MIN : REAL ;
  IN_MAX : REAL ;
  OUT_MIN : REAL ;
  OUT_MAX : REAL ;
END_VAR
VAR_OUTPUT
  OUT : REAL ;
  ERROR : BOOL ;
END_VAR
VAR_TEMP
  Diff : REAL ;
  IN : INT ;
  IN_REAL : REAL ;
END_VAR
BEGIN
// body was compiled from an SCL source; compiled code not shown
END_FUNCTION

FUNCTION "fnWordPack" : VOID	// FC 2
VERSION : 0.0
VAR_INPUT
  bHigh : BYTE ;
  bLow : BYTE ;
END_VAR
VAR_OUTPUT
  OUT : WORD ;
END_VAR
VAR_TEMP
  iTemp : INT ;
END_VAR
BEGIN
// body was compiled from an SCL source; compiled code not shown
END_FUNCTION

FUNCTION "fnBytesToReal" : VOID	// FC 3
VERSION : 0.0
VAR_INPUT
  bHigh : BYTE ;
  bLow : BYTE ;
END_VAR
VAR_OUTPUT
  OUT : REAL ;
END_VAR
VAR_TEMP
  iTemp : INT ;
END_VAR
BEGIN
// body was compiled from an SCL source; compiled code not shown
END_FUNCTION

FUNCTION "fnBytesToRealOneComma" : VOID	// FC 4
VERSION : 0.0
VAR_INPUT
  bHigh : BYTE ;
  bLow : BYTE ;
END_VAR
VAR_OUTPUT
  OUT : REAL ;
END_VAR
VAR_TEMP
  iTemp : INT ;
END_VAR
BEGIN
// body was compiled from an SCL source; compiled code not shown
END_FUNCTION

FUNCTION "fnBytesToRealPressure" : VOID	// FC 5
VERSION : 0.0
VAR_INPUT
  bHigh : BYTE ;
  bLow : BYTE ;
END_VAR
VAR_OUTPUT
  OUT : REAL ;
END_VAR
VAR_TEMP
  iTemp : INT ;
END_VAR
BEGIN
// body was compiled from an SCL source; compiled code not shown
END_FUNCTION

FUNCTION "fnBytesToRealTwoComas" : VOID	// FC 6
VERSION : 0.0
VAR_INPUT
  bHigh : BYTE ;
  bLow : BYTE ;
END_VAR
VAR_OUTPUT
  OUT : REAL ;
END_VAR
VAR_TEMP
  iTemp : INT ;
END_VAR
BEGIN
// body was compiled from an SCL source; compiled code not shown
END_FUNCTION

FUNCTION "StartStopByte" : VOID	// FC 7
VERSION : 0.0
VAR_INPUT
  xStart : BOOL ;
  xStop : BOOL ;
END_VAR
VAR_OUTPUT
  OUT : BYTE ;
END_VAR
VAR_TEMP
  iTemp : INT ;
END_VAR
BEGIN
// body was compiled from an SCL source; compiled code not shown
END_FUNCTION

FUNCTION "LinTrafoInt" : VOID	// FC 8
VERSION : 0.0
VAR_INPUT
  IN : INT ;
  IN_MIN : REAL ;
  IN_MAX : REAL ;
  OUT_MIN : REAL ;
  OUT_MAX : REAL ;
END_VAR
VAR_OUTPUT
  OUT : REAL ;
  ERROR : BOOL ;
END_VAR
VAR_TEMP
  Diff : REAL ;
  IN_REAL : REAL ;
END_VAR
BEGIN
// body was compiled from an SCL source; compiled code not shown
END_FUNCTION

FUNCTION "ByteToByte" : VOID	// FC 9
VERSION : 0.0
VAR_INPUT
  bIn : BYTE ;
END_VAR
VAR_OUTPUT
  OUT : BYTE ;
END_VAR
BEGIN
// body was compiled from an SCL source; compiled code not shown
END_FUNCTION

DATA_BLOCK "GLV"	// DB 1
VERSION : 0.1
  STRUCT
   Her : INT ;	//Temporary placeholder variable
   CompressedAirPressureAft : BOOL ;
  END_STRUCT ;	
BEGIN
END_DATA_BLOCK

DATA_BLOCK "A_Sensors"	// DB 2
VERSION : 0.1
  STRUCT
   KB_1_1_1PIR7 : REAL  := 1.000000e+001;	//CompressedAirPressureAfterKB_1_1
   KB_1_2_2PIR7 : REAL ;	//CompressedAirPressureAfter_KB_1_2
   KZA_1_1_1PIR6 : REAL ;	//N_PressureAfter_KZA_1_1
   KZA_1_2_2PIR6 : REAL ;	//CompressedAirPressureAfter
   KB_2_PIR8 : REAL ;	//CompressedAirPressureAfter_KB_2
   KZA_2_2_2PIR20 : REAL ;	//N_PressureAfter_KZA_2_2
   TIR10 : REAL ;	//N_PressureIntoSystem
   FIR10 : REAL ;	//N_Consume
   PIR5 : REAL ;	//N_PressureIntoSystem
   FIR5 : REAL ;	//N_ConsumeSystem
   PIRC21 : REAL ;	//N_PressureDiagn
   One_PIR27 : REAL ;	//N_PressureAfter_PB_2_1
   QIRAH3 : REAL ;	//O2_Consis_KZA_1_1_2
   Two_PIR27 : REAL ;	//AirPressure_PB_2_2
   PIR4 : REAL ;	//AirPressure_
   FIR_4 : REAL ;	//CompressedAirConsum
   PIRC22 : REAL ;	//AirPressure
   PIRC23 : REAL ;	//AirPressure_PBT_1
   PIRC24 : REAL ;	//AirPressure_PBK_1
   PIRC25 : REAL ;	//AirPressure
   FIR_25 : REAL ;	//CompressedAirConsum
   One_PIRC26 : REAL ;	//AirPressure_PB_1_1
   Two_PIRC26 : REAL ;	//AirPressure_PB_1_2
   PIRC_C10 : REAL ;	//N_Temp
   TIR5 : REAL ;	//N_Temp
   TIR4 : REAL ;	//Air_Temp
   TIR25 : REAL ;	//Air_Temp
   AIR1 : REAL ;	//Air_Wetness
   One_PIR20 : REAL ;
   Qirahq4 : REAL ;
  END_STRUCT ;	
BEGIN
END_DATA_BLOCK

DATA_BLOCK "DI"	// DB 3
VERSION : 0.1
  STRUCT
   DI_XL1_QL3 : BOOL ;
   DI_XL2_QL3 : BOOL ;
   DI_Q3_Bad : BOOL ;
   DI_AB1_Working : BOOL ;
   DI_Kb_1_1_Working : BOOL ;
   DI_Kb_1_1_Alm : BOOL ;
   DI_Kb_1_2_Working : BOOL ;
   DI_Kb_1_2_Alm : BOOL ;
   DI_Kb_2_Working : BOOL ;
   DI_Kb_2_Alm : BOOL ;
   DI_Kd_1_Working : BOOL ;
   DI_Kd_1_Alm : BOOL ;
   DI_ZB_1_Opn : BOOL ;
   DI_ZB_1_Cls : BOOL ;
   DI_ZB_1_Local : BOOL ;
   DI_ZB_1_Alm : BOOL ;
   DI_ZB_2_Opn : BOOL ;
   DI_ZB_2_Cls : BOOL ;
   DI_ZB_2_Local : BOOL ;
   DI_ZB_2_Alm : BOOL ;
   DI_ZB_3_Opn : BOOL ;
   DI_ZB_3_Cls : BOOL ;
   DI_ZB_3_Local : BOOL ;
   DI_ZB_3_Alm : BOOL ;
   DI_EUV_001_Opn : BOOL ;
   DI_EUV_001_Cls : BOOL ;
   DI_EUV_001_Local : BOOL ;
   DI_EUV_001_Alm : BOOL ;
   DI_EUV_002_Opn : BOOL ;
   DI_EUV_002_Cls : BOOL ;
   DI_EUV_002_Local : BOOL ;
   DI_EUV_002_Alm : BOOL ;
   DI_EUV_003_Opn : BOOL ;
   DI_EUV_003_Cls : BOOL ;
   DI_EUV_003_Local : BOOL ;
   DI_EUV_003_Alm : BOOL ;
   DI_KZA_1_1_QSA1_1_QSL1_1 : BOOL ;
   DI_KZA_1_1_QSA1_1_QSL1_2 : BOOL ;
   DI_KZA_1_1_QSA1_1_QSL2_1 : BOOL ;
   DI_KZA_1_1_QSA1_1_QSL2_2 : BOOL ;
   DI_KZA_1_1_QSA1_1_QSL3_1 : BOOL ;
   DI_KZA_1_1_QSA1_1_QSL3_2 : BOOL ;
   DI_KZA_1_1_QSA1_1_QSL4_1 : BOOL ;
   DI_KZA_1_1_QSA1_1_QSL4_2 : BOOL ;
   DI_KD_1_QSA_1_5QSL1_5_1 : BOOL ;
   DI_KD_1_QSA_1_5QSL1_5_2 : BOOL ;
   DI_Q3_BAD_1 : BOOL ;
   DI_AB1_XLA_AV1_Alm : BOOL ;
   DI_AB2_XL_AV2_Working : BOOL ;
   DI_AB2_XLA_AV2_Alm : BOOL ;
   DI_AB3_XL_AV3_Working : BOOL ;
   DI_AB3_XLA_AV3_Alm : BOOL ;
   DI_AB4_XL_AV4_Working : BOOL ;
   DI_AB4_XLA_AV4_Alm : BOOL ;
   DI_P2_XLP_2_Working : BOOL ;
   DI_P2_XLP_2_Alm : BOOL ;
   DI_P3_XLP_3_Working : BOOL ;
   DI_P3_XLP_3_Alm : BOOL ;
   DI_IBP_1_Working : BOOL ;
   DI_IBP_1_Alm : BOOL ;
   DI_IBP_1_Bypass : BOOL ;
   DI_IBP_2_Working : BOOL ;
   DI_IBP_2_Alm : BOOL ;
   DI_IBP_2_Bypass : BOOL ;
  END_STRUCT ;	
BEGIN
END_DATA_BLOCK

DATA_BLOCK "SensorsSettings"	// DB 4
VERSION : 0.1
  STRUCT
   One_PIR7_Min : REAL  := 1.000000e+001;	//CompressedAirPressureAfter_KB_1_1
   One_PIR7_Max : REAL ;	//CompressedAirPressureAfter_KB_1_1
   Two_PIR7_Min : REAL ;	//CompressedAirPressureAfter_KB_1_2
   Two_PIR7_Max : REAL ;	//CompressedAirPressureAfter_KB_1_2
   One_PIR6_Min : REAL ;	//N_PressureAfter_KZA_1_1
   One_PIR6_Max : REAL ;	//N_PressureAfter_KZA_1_1
   Two_PIR6_Min : REAL ;	//N_PressureAfter_KZA_1_2
   Two_PIR6_Max : REAL ;	//N_PressureAfter_KZA_1_2
   PIR8_Min : REAL ;	//CompressedAirPressureAfter_KB_2
   PIR8_Max : REAL ;	//CompressedAirPressureAfter_KB_2
   Two_PIR20_Min : REAL ;	//N_PressureAfter_KZA_2_2
   Two_PIR20_Max : REAL ;	//N_PressureAfter_KZA_2_2
   TIR10_Min : REAL ;	//N_PressureIntoSystem
   TIR10_Max : REAL ;	//N_PressureIntoSystem
   FIR10_Min : REAL ;	//N_Consume
   FIR10_Max : REAL ;	//N_Consume
   PIR5_Min : REAL ;	//N_PressureIntoSystem
   PIR5_Max : REAL ;	//N_PressureIntoSystem
   FIR5_Min : REAL ;	//N_ConsumeSystem
   FIR5_Max : REAL ;	//N_ConsumeSystem
   PIRC21_Min : REAL ;	//N_PressureDiagn
   PIRC21_Max : REAL ;	//N_PressureDiagn
   One_PIR27_Min : REAL ;	//N_PressureAfter_PB_2_1
   One_PIR27_Max : REAL ;	//N_PressureAfter_PB_2_1
   QIRAH3_Min : REAL ;	//O2_Consis_KZA_1_1_2
   QIRAH3_Max : REAL ;	//O2_Consis_KZA_1_1_2
   Two_PIR27_Min : REAL ;	//AirPressure_PB_2_2
   Two_PIR27_Max : REAL ;	//AirPressure_PB_2_2
   PIR4_Min : REAL ;	//AirPressure
   PIR4_Max : REAL ;	//AirPressure
   FIR_4_Min : REAL ;	//CompressedAirConsum
   FIR_4_Max : REAL ;	//CompressedAirConsum
   PIRC22_Min : REAL ;	//AirPressure_PIRC22
   PIRC22_Max : REAL ;	//AirPressure_PIRC22
   PIRC23_Min : REAL ;	//AirPressure_PBT_1
   PIRC23_Max : REAL ;	//AirPressure_PBT_1
   PIRC24_Min : REAL ;	//AirPressure_PBK_1
   PIRC24_Max : REAL ;	//AirPressure_PBK_1
   PIRC25_Min : REAL ;	//AirPressure
   PIRC25_Max : REAL ;	//AirPressure
   FIR_25_Min : REAL ;	//CompressedAirConsum
   FIR_25_Max : REAL ;	//CompressedAirConsum
   One_PIRC26_Min : REAL ;	//AirPressure_PB_1_1
   One_PIRC26_Max : REAL ;	//AirPressure_PB_1_1
   Two_PIRC26_Min : REAL ;	//AirPressure_PB_1_2
   Two_PIRC26_Max : REAL ;	//AirPressure_PB_1_2
   PIRC_C10_Min : REAL ;	//N_Temp
   PIRC_C10_Max : REAL ;	//N_Temp
   TIR5_Min : REAL ;	//N_Temp
   TIR5_Max : REAL ;	//N_Temp
   TIR4_Min : REAL ;	//Air_Temp
   TIR4_Max : REAL ;	//Air_Temp
   TIR25_Min : REAL ;	//Air_Temp
   TIR25_Max : REAL ;	//Air_Temp
   AIR1_Min : REAL ;	//Air_Wetness_AIR1
   AIR1_Max : REAL ;	//Air_Wetness_AIR1
   One_PIR20_Min : REAL ;	//N_PressureAfter_KZA_2_2
   One_PIR20_Max : REAL ;	//N_PressureAfter_KZA_2_2
   QIRAH4H4_Min : REAL ;
   QIRAH4H4_Max : REAL ;
  END_STRUCT ;	
BEGIN
END_DATA_BLOCK

DATA_BLOCK "Valves"	// DB 5
VERSION : 0.1
  STRUCT
   xOnAuto_KB_1_1 : BOOL ;	//Temporary placeholder variable
   xOnAuto_KB_1_2 : BOOL ;
   xOnAuto_KB_2 : BOOL ;
   xOnAuto_KD_1 : BOOL ;
   xOnAuto_ZB_1 : BOOL ;
   xOnAuto_ZB_2 : BOOL ;
   xOnAuto_ZB_3 : BOOL ;
   xOnManual_KB_1_1 : BOOL ;
   xOnManual_KB_1_2 : BOOL ;
   xOnManual_KB_2 : BOOL ;
   xOnManual_KD_1 : BOOL ;
   xOnManual_ZB_1 : BOOL ;
   xOnManual_ZB_2 : BOOL ;
   xOnManual_ZB_3 : BOOL ;
   xManualMode_KB_1_1 : BOOL ;
   xManualMode_KB_1_2 : BOOL ;
   xManualMode_KB_2 : BOOL ;
   xManualMode_KD_1 : BOOL ;
   xManualMode_ZB_1 : BOOL ;
   xManualMode_ZB_2 : BOOL ;
   xManualMode_ZB_3 : BOOL ;
   xStop_KB_1_1 : BOOL ;
   xStop_KB_1_2 : BOOL ;
   xStop_KB_2 : BOOL ;
   xStop_KD_1 : BOOL ;
   xStop_ZB_1 : BOOL ;
   xStop_ZB_2 : BOOL ;
   xStop_ZB_3 : BOOL ;
   wState_ZB_1 : INT ;
   wState_ZB_2 : INT ;
   wState_ZB_3 : INT ;
   xOffAuto_ZB_1 : BOOL ;
   xOffAuto_ZB_2 : BOOL ;
   xOffAuto_ZB_3 : BOOL ;
   xOffAuto_ZB_4 : BOOL ;
   xOffManual_ZB_1 : BOOL ;
   xOffManual_ZB_2 : BOOL ;
   xOffManual_ZB_3 : BOOL ;
   xOffManual_ZB_4 : BOOL ;
   xOnAuto_ZB_4 : BOOL ;
   xOnManual_ZB_4 : BOOL ;
   xStop_ZB_4 : BOOL ;
   xStop_ManualZB_1 : BOOL ;
   xStop_ManualZB_2 : BOOL ;
   xStop_ManualZB_3 : BOOL ;
   xStop_ManualZB_4 : BOOL ;
  END_STRUCT ;	
BEGIN
END_DATA_BLOCK

DATA_BLOCK "BD_Coils"	// DB 6
VERSION : 0.1
  STRUCT
   B_0 : BYTE ;
   B_1 : BYTE ;
   Running_Stopped : BOOL ;
   Load_Unload : BOOL ;
   General_Warning : BOOL ;
   GeneralShutdownWarning : BOOL ;
   GeneralShutdown : BOOL ;
   GeneralService : BOOL ;
   GeneralStartFailure : BOOL ;
   EmergencyStop : BOOL ;
   Automatic_Manual : BOOL ;
   Remote_Local : BOOL ;
  END_STRUCT ;	
BEGIN
END_DATA_BLOCK

DATA_BLOCK "KB1_1_Coils"	// DB 7
VERSION : 0.1
  STRUCT
   B_0 : BYTE ;
   B_1 : BYTE ;
   Running_Stopped : BOOL ;
   Load_Unload : BOOL ;
   General_Warning : BOOL ;
   GeneralShutdownWarning : BOOL ;
   GeneralShutdown : BOOL ;
   GeneralService : BOOL ;
   GeneralStartFailure : BOOL ;
   EmergencyStop : BOOL ;
   Automatic_Manual : BOOL ;
   Remote_Local : BOOL ;
  END_STRUCT ;	
BEGIN
END_DATA_BLOCK

DATA_BLOCK "KB1_2_Coils"	// DB 8
VERSION : 0.1
  STRUCT
   B_0 : BYTE ;
   B_1 : BYTE ;
   Running_Stopped : BOOL ;
   Load_Unload : BOOL ;
   General_Warning : BOOL ;
   GeneralShutdownWarning : BOOL ;
   GeneralShutdown : BOOL ;
   GeneralService : BOOL ;
   GeneralStartFailure : BOOL ;
   EmergencyStop : BOOL ;
   Automatic_Manual : BOOL ;
   Remote_Local : BOOL ;
   DB_VAR : INT ;	//Temporary placeholder variable
  END_STRUCT ;	
BEGIN
END_DATA_BLOCK

DATA_BLOCK "KB2_Coils"	// DB 9
VERSION : 0.1
  STRUCT
   B_0 : BYTE ;
   B_1 : BYTE ;
   Running_Stopped : BOOL ;
   Load_Unload : BOOL ;
   General_Warning : BOOL ;
   GeneralShutdownWarning : BOOL ;
   GeneralShutdown : BOOL ;
   GeneralService : BOOL ;
   GeneralStartFailure : BOOL ;
   EmergencyStop : BOOL ;
   Automatic_Manual : BOOL ;
   Remote_Local : BOOL ;
  END_STRUCT ;	
BEGIN
END_DATA_BLOCK

DATA_BLOCK "PO1_1_Coils"	// DB 10
VERSION : 0.1
  STRUCT
   B_0 : BYTE ;
   B_1 : BYTE ;
   Running_Stopped : BOOL ;
   Load_Unload : BOOL ;
   General_Warning : BOOL ;
   GeneralShutdownWarning : BOOL ;
   GeneralShutdown : BOOL ;
   GeneralService : BOOL ;
   GeneralStartFailure : BOOL ;
   EmergencyStop : BOOL ;
   Automatic_Manual : BOOL ;
   Remote_Local : BOOL ;
  END_STRUCT ;	
BEGIN
END_DATA_BLOCK

DATA_BLOCK "PO1_2_Coils"	// DB 11
VERSION : 0.1
  STRUCT
   B_0 : BYTE ;
   B_1 : BYTE ;
   Running_Stopped : BOOL ;
   Load_Unload : BOOL ;
   General_Warning : BOOL ;
   GeneralShutdownWarning : BOOL ;
   GeneralShutdown : BOOL ;
   GeneralService : BOOL ;
   GeneralStartFailure : BOOL ;
   EmergencyStop : BOOL ;
   Automatic_Manual : BOOL ;
   Remote_Local : BOOL ;
  END_STRUCT ;	
BEGIN
END_DATA_BLOCK

DATA_BLOCK "GA1_1_Coils"	// DB 12
VERSION : 0.1
  STRUCT
   B_0 : BYTE ;
   B_1 : BYTE ;
   Running_Stopped : BOOL ;
   Load_Unload : BOOL ;
   General_Warning : BOOL ;
   GeneralShutdownWarning : BOOL ;
   GeneralShutdown : BOOL ;
   GeneralService : BOOL ;
   GeneralStartFailure : BOOL ;
   EmergencyStop : BOOL ;
   Automatic_Manual : BOOL ;
   Remote_Local : BOOL ;
  END_STRUCT ;	
BEGIN
END_DATA_BLOCK

DATA_BLOCK "GA1_2_Coils"	// DB 13
VERSION : 0.1
  STRUCT
   B_0 : BYTE ;
   B_1 : BYTE ;
   Running_Stopped : BOOL ;
   Load_Unload : BOOL ;
   General_Warning : BOOL ;
   GeneralShutdownWarning : BOOL ;
   GeneralShutdown : BOOL ;
   GeneralService : BOOL ;
   GeneralStartFailure : BOOL ;
   EmergencyStop : BOOL ;
   Automatic_Manual : BOOL ;
   Remote_Local : BOOL ;
  END_STRUCT ;	
BEGIN
END_DATA_BLOCK

DATA_BLOCK "GA2_1_Coils"	// DB 14
VERSION : 0.1
  STRUCT
   B_0 : BYTE ;
   B_1 : BYTE ;
   Running_Stopped : BOOL ;
   Load_Unload : BOOL ;
   General_Warning : BOOL ;
   GeneralShutdownWarning : BOOL ;
   GeneralShutdown : BOOL ;
   GeneralService : BOOL ;
   GeneralStartFailure : BOOL ;
   EmergencyStop : BOOL ;
   Automatic_Manual : BOOL ;
   Remote_Local : BOOL ;
  END_STRUCT ;	
BEGIN
END_DATA_BLOCK

DATA_BLOCK "GA2_2_Coils"	// DB 15
VERSION : 0.1
  STRUCT
   B_0 : BYTE ;
   B_1 : BYTE ;
   Running_Stopped : BOOL ;
   Load_Unload : BOOL ;
   General_Warning : BOOL ;
   GeneralShutdownWarning : BOOL ;
   GeneralShutdown : BOOL ;
   GeneralService : BOOL ;
   GeneralStartFailure : BOOL ;
   EmergencyStop : BOOL ;
   Automatic_Manual : BOOL ;
   Remote_Local : BOOL ;
  END_STRUCT ;	
BEGIN
END_DATA_BLOCK

DATA_BLOCK "BD_AI_1"	// DB 16
VERSION : 0.1
  STRUCT
   B_0 : BYTE ;
   B_1 : BYTE ;
   B_2 : BYTE ;
   B_3 : BYTE ;
   B_4 : BYTE ;
   B_5 : BYTE ;
   B_6 : BYTE ;
   B_7 : BYTE ;
   B_8 : BYTE ;
  END_STRUCT ;	
BEGIN
END_DATA_BLOCK

DATA_BLOCK "KB1_1_AI_1"	// DB 17
VERSION : 0.1
  STRUCT
   B_0 : BYTE ;
   B_1 : BYTE ;
   B_2 : BYTE ;
   B_3 : BYTE ;
   B_4 : BYTE ;
   B_5 : BYTE ;
   B_6 : BYTE ;
   B_7 : BYTE ;
   B_8 : BYTE ;
   B_9 : BYTE ;
   B_10 : BYTE ;
   B_11 : BYTE ;
   B_12 : BYTE ;
   B_13 : BYTE ;
   B_14 : BYTE ;
   B_15 : BYTE ;
   B_16 : BYTE ;
  END_STRUCT ;	
BEGIN
END_DATA_BLOCK

DATA_BLOCK "KB1_1_AI_2"	// DB 18
VERSION : 0.1
  STRUCT
   B_0 : BYTE ;
   B_1 : BYTE ;
   B_2 : BYTE ;
   B_3 : BYTE ;
   B_4 : BYTE ;
   B_5 : BYTE ;
   B_6 : BYTE ;
   B_7 : BYTE ;
   B_8 : BYTE ;
   B_9 : BYTE ;
   B_10 : BYTE ;
   B_11 : BYTE ;
   B_12 : BYTE ;
   B_13 : BYTE ;
   B_14 : BYTE ;
   B_15 : BYTE ;
   B_16 : BYTE ;
   B_17 : BYTE ;
   B_18 : BYTE ;
   B_19 : BYTE ;
   B_20 : BYTE ;
   B_21 : BYTE ;
   B_22 : BYTE ;
   B_23 : BYTE ;
   B_24 : BYTE ;
   B_25 : BYTE ;
   B_26 : BYTE ;
   B_27 : BYTE ;
   B_28 : BYTE ;
   B_29 : BYTE ;
   B_30 : BYTE ;
   B_31 : BYTE ;
   B_32 : BYTE ;
  END_STRUCT ;	
BEGIN
END_DATA_BLOCK

DATA_BLOCK "KB1_1_AI_3"	// DB 19
VERSION : 0.1
  STRUCT
   B_0 : BYTE ;
   B_1 : BYTE ;
   B_2 : BYTE ;
   B_3 : BYTE ;
   B_4 : BYTE ;
   B_5 : BYTE ;
   B_6 : BYTE ;
   B_7 : BYTE ;
   B_8 : BYTE ;
   B_9 : BYTE ;
   B_10 : BYTE ;
   B_11 : BYTE ;
   B_12 : BYTE ;
   B_13 : BYTE ;
  END_STRUCT ;	
BEGIN
END_DATA_BLOCK

DATA_BLOCK "KB1_2_AI_1"	// DB 20
VERSION : 0.1
  STRUCT
   B_0 : BYTE ;
   B_1 : BYTE ;
   B_2 : BYTE ;
   B_3 : BYTE ;
   B_4 : BYTE ;
   B_5 : BYTE ;
   B_6 : BYTE ;
   B_7 : BYTE ;
   B_8 : BYTE ;
   B_9 : BYTE ;
   B_10 : BYTE ;
   B_11 : BYTE ;
   B_12 : BYTE ;
   B_13 : BYTE ;
   B_14 : BYTE ;
   B_15 : BYTE ;
   B_16 : BYTE ;
  END_STRUCT ;	
BEGIN
END_DATA_BLOCK

DATA_BLOCK "KB1_2_AI_2"	// DB 21
VERSION : 0.1
  STRUCT
   B_0 : BYTE ;
   B_1 : BYTE ;
   B_2 : BYTE ;
   B_3 : BYTE ;
   B_4 : BYTE ;
   B_5 : BYTE ;
   B_6 : BYTE ;
   B_7 : BYTE ;
   B_8 : BYTE ;
   B_9 : BYTE ;
   B_10 : BYTE ;
   B_11 : BYTE ;
   B_12 : BYTE ;
   B_13 : BYTE ;
   B_14 : BYTE ;
   B_15 : BYTE ;
   B_16 : BYTE ;
   B_17 : BYTE ;
   B_18 : BYTE ;
   B_19 : BYTE ;
   B_20 : BYTE ;
   B_21 : BYTE ;
   B_22 : BYTE ;
   B_23 : BYTE ;
   B_24 : BYTE ;
   B_25 : BYTE ;
   B_26 : BYTE ;
   B_27 : BYTE ;
   B_28 : BYTE ;
   B_29 : BYTE ;
   B_30 : BYTE ;
   B_31 : BYTE ;
   B_32 : BYTE ;
  END_STRUCT ;	
BEGIN
END_DATA_BLOCK

DATA_BLOCK "KB1_2_AI_3"	// DB 22
VERSION : 0.1
  STRUCT
   B_0 : BYTE ;
   B_1 : BYTE ;
   B_2 : BYTE ;
   B_3 : BYTE ;
   B_4 : BYTE ;
   B_5 : BYTE ;
   B_6 : BYTE ;
   B_7 : BYTE ;
   B_8 : BYTE ;
   B_9 : BYTE ;
   B_10 : BYTE ;
   B_11 : BYTE ;
   B_12 : BYTE ;
   B_13 : BYTE ;
  END_STRUCT ;	
BEGIN
END_DATA_BLOCK

DATA_BLOCK "KB2_AI_1"	// DB 23
VERSION : 0.1
  STRUCT
   B_0 : BYTE ;
   B_1 : BYTE ;
   B_2 : BYTE ;
   B_3 : BYTE ;
   B_4 : BYTE ;
   B_5 : BYTE ;
   B_6 : BYTE ;
   B_7 : BYTE ;
   B_8 : BYTE ;
   B_9 : BYTE ;
   B_10 : BYTE ;
   B_11 : BYTE ;
   B_12 : BYTE ;
   B_13 : BYTE ;
   B_14 : BYTE ;
   B_15 : BYTE ;
   B_16 : BYTE ;
  END_STRUCT ;	
BEGIN
END_DATA_BLOCK

DATA_BLOCK "KB2_AI_2"	// DB 24
VERSION : 0.1
  STRUCT
   B_0 : BYTE ;
   B_1 : BYTE ;
   B_2 : BYTE ;
   B_3 : BYTE ;
   B_4 : BYTE ;
   B_5 : BYTE ;
   B_6 : BYTE ;
   B_7 : BYTE ;
   B_8 : BYTE ;
   B_9 : BYTE ;
   B_10 : BYTE ;
   B_11 : BYTE ;
   B_12 : BYTE ;
   B_13 : BYTE ;
   B_14 : BYTE ;
   B_15 : BYTE ;
   B_16 : BYTE ;
   B_17 : BYTE ;
   B_18 : BYTE ;
   B_19 : BYTE ;
   B_20 : BYTE ;
   B_21 : BYTE ;
   B_22 : BYTE ;
   B_23 : BYTE ;
   B_24 : BYTE ;
   B_25 : BYTE ;
   B_26 : BYTE ;
   B_27 : BYTE ;
   B_28 : BYTE ;
  END_STRUCT ;	
BEGIN
END_DATA_BLOCK

DATA_BLOCK "KB2_AI_3"	// DB 25
VERSION : 0.1
  STRUCT
   B_0 : BYTE ;
   B_1 : BYTE ;
   B_2 : BYTE ;
   B_3 : BYTE ;
   B_4 : BYTE ;
   B_5 : BYTE ;
   B_6 : BYTE ;
   B_7 : BYTE ;
   B_8 : BYTE ;
   B_9 : BYTE ;
   B_10 : BYTE ;
   B_11 : BYTE ;
   B_12 : BYTE ;
   B_13 : BYTE ;
   B_14 : BYTE ;
   B_15 : BYTE ;
   B_16 : BYTE ;
   B_17 : BYTE ;
   B_18 : BYTE ;
   B_19 : BYTE ;
   B_20 : BYTE ;
  END_STRUCT ;	
BEGIN
END_DATA_BLOCK

DATA_BLOCK "KB2_AI_4"	// DB 26
VERSION : 0.1
  STRUCT
   B_0 : BYTE ;
   B_1 : BYTE ;
   B_2 : BYTE ;
   B_3 : BYTE ;
   B_4 : BYTE ;
   B_5 : BYTE ;
   B_6 : BYTE ;
   B_7 : BYTE ;
   B_8 : BYTE ;
   B_9 : BYTE ;
   B_10 : BYTE ;
   B_11 : BYTE ;
   B_12 : BYTE ;
   B_13 : BYTE ;
   B_14 : BYTE ;
   B_15 : BYTE ;
   B_16 : BYTE ;
   B_17 : BYTE ;
   B_18 : BYTE ;
   B_19 : BYTE ;
   B_20 : BYTE ;
   B_21 : BYTE ;
   B_22 : BYTE ;
   B_23 : BYTE ;
   B_24 : BYTE ;
  END_STRUCT ;	
BEGIN
END_DATA_BLOCK

DATA_BLOCK "PO1_1_AI"	// DB 27
VERSION : 0.1
  STRUCT
   B_0 : BYTE ;
   B_1 : BYTE ;
   B_2 : BYTE ;
   B_3 : BYTE ;
   B_4 : BYTE ;
   B_5 : BYTE ;
   B_6 : BYTE ;
   B_7 : BYTE ;
   B_8 : BYTE ;
   B_9 : BYTE ;
   B_10 : BYTE ;
   B_11 : BYTE ;
   B_12 : BYTE ;
   B_13 : BYTE ;
   B_14 : BYTE ;
   B_15 : BYTE ;
   B_16 : BYTE ;
   B_17 : BYTE ;
   B_18 : BYTE ;
   B_19 : BYTE ;
   B_20 : BYTE ;
   B_21 : BYTE ;
   B_22 : BYTE ;
   B_23 : BYTE ;
   B_24 : BYTE ;
   B_25 : BYTE ;
   B_26 : BYTE ;
   B_27 : BYTE ;
   B_28 : BYTE ;
   B_29 : BYTE ;
   B_30 : BYTE ;
   B_31 : BYTE ;
   B_32 : BYTE ;
   B_33 : BYTE ;
   B_34 : BYTE ;
   B_35 : BYTE ;
   B_36 : BYTE ;
   B_37 : BYTE ;
   B_38 : BYTE ;
   B_39 : BYTE ;
   B_40 : BYTE ;
   B_41 : BYTE ;
   B_42 : BYTE ;
   B_43 : BYTE ;
   B_44 : BYTE ;
  END_STRUCT ;	
BEGIN
END_DATA_BLOCK

DATA_BLOCK "PO1_2_AI"	// DB 28
VERSION : 0.1
  STRUCT
   B_0 : BYTE ;
   B_1 : BYTE ;
   B_2 : BYTE ;
   B_3 : BYTE ;
   B_4 : BYTE ;
   B_5 : BYTE ;
   B_6 : BYTE ;
   B_7 : BYTE ;
   B_8 : BYTE ;
   B_9 : BYTE ;
   B_10 : BYTE ;
   B_11 : BYTE ;
   B_12 : BYTE ;
   B_13 : BYTE ;
   B_14 : BYTE ;
   B_15 : BYTE ;
   B_16 : BYTE ;
   B_17 : BYTE ;
   B_18 : BYTE ;
   B_19 : BYTE ;
   B_20 : BYTE ;
   B_21 : BYTE ;
   B_22 : BYTE ;
   B_23 : BYTE ;
   B_24 : BYTE ;
   B_25 : BYTE ;
   B_26 : BYTE ;
   B_27 : BYTE ;
   B_28 : BYTE ;
   B_29 : BYTE ;
   B_30 : BYTE ;
   B_31 : BYTE ;
   B_32 : BYTE ;
   B_33 : BYTE ;
   B_34 : BYTE ;
   B_35 : BYTE ;
   B_36 : BYTE ;
   B_37 : BYTE ;
   B_38 : BYTE ;
   B_39 : BYTE ;
   B_40 : BYTE ;
   B_41 : BYTE ;
   B_42 : BYTE ;
   B_43 : BYTE ;
   B_44 : BYTE ;
  END_STRUCT ;	
BEGIN
END_DATA_BLOCK

DATA_BLOCK "GA1_1_AI_1"	// DB 29
VERSION : 0.1
  STRUCT
   B_0 : BYTE ;
   B_1 : BYTE ;
   B_2 : BYTE ;
   B_3 : BYTE ;
   B_4 : BYTE ;
   B_5 : BYTE ;
   B_6 : BYTE ;
   B_7 : BYTE ;
   B_8 : BYTE ;
   B_9 : BYTE ;
   B_10 : BYTE ;
   B_11 : BYTE ;
   B_12 : BYTE ;
   B_13 : BYTE ;
   B_14 : BYTE ;
   B_15 : BYTE ;
   B_16 : BYTE ;
   B_17 : BYTE ;
   B_18 : BYTE ;
   B_19 : BYTE ;
   B_20 : BYTE ;
  END_STRUCT ;	
BEGIN
END_DATA_BLOCK

DATA_BLOCK "GA1_1_AI_2"	// DB 30
VERSION : 0.1
  STRUCT
   B_0 : BYTE ;
   B_1 : BYTE ;
   B_2 : BYTE ;
   B_3 : BYTE ;
   B_4 : BYTE ;
   B_5 : BYTE ;
   B_6 : BYTE ;
   B_7 : BYTE ;
   B_8 : BYTE ;
   B_9 : BYTE ;
   B_10 : BYTE ;
   B_11 : BYTE ;
   B_12 : BYTE ;
   B_13 : BYTE ;
   B_14 : BYTE ;
   B_15 : BYTE ;
   B_16 : BYTE ;
  END_STRUCT ;	
BEGIN
END_DATA_BLOCK

DATA_BLOCK "GA1_2_AI_1"	// DB 31
VERSION : 0.1
  STRUCT
   B_0 : BYTE ;
   B_1 : BYTE ;
   B_2 : BYTE ;
   B_3 : BYTE ;
   B_4 : BYTE ;
   B_5 : BYTE ;
   B_6 : BYTE ;
   B_7 : BYTE ;
   B_8 : BYTE ;
   B_9 : BYTE ;
   B_10 : BYTE ;
   B_11 : BYTE ;
   B_12 : BYTE ;
   B_13 : BYTE ;
   B_14 : BYTE ;
   B_15 : BYTE ;
   B_16 : BYTE ;
   B_17 : BYTE ;
   B_18 : BYTE ;
   B_19 : BYTE ;
   B_20 : BYTE ;
  END_STRUCT ;	
BEGIN
END_DATA_BLOCK

DATA_BLOCK "GA1_2_AI_2"	// DB 32
VERSION : 0.1
  STRUCT
   B_0 : BYTE ;
   B_1 : BYTE ;
   B_2 : BYTE ;
   B_3 : BYTE ;
   B_4 : BYTE ;
   B_5 : BYTE ;
   B_6 : BYTE ;
   B_7 : BYTE ;
   B_8 : BYTE ;
   B_9 : BYTE ;
   B_10 : BYTE ;
   B_11 : BYTE ;
   B_12 : BYTE ;
   B_13 : BYTE ;
   B_14 : BYTE ;
   B_15 : BYTE ;
   B_16 : BYTE ;
  END_STRUCT ;	
BEGIN
END_DATA_BLOCK

DATA_BLOCK "GA2_1_AI_1"	// DB 33
VERSION : 0.1
  STRUCT
   B_0 : BYTE ;
   B_1 : BYTE ;
   B_2 : BYTE ;
   B_3 : BYTE ;
   B_4 : BYTE ;
   B_5 : BYTE ;
   B_6 : BYTE ;
   B_7 : BYTE ;
   B_8 : BYTE ;
   B_9 : BYTE ;
   B_10 : BYTE ;
   B_11 : BYTE ;
   B_12 : BYTE ;
   B_13 : BYTE ;
   B_14 : BYTE ;
   B_15 : BYTE ;
   B_16 : BYTE ;
   B_17 : BYTE ;
   B_18 : BYTE ;
   B_19 : BYTE ;
   B_20 : BYTE ;
  END_STRUCT ;	
BEGIN
END_DATA_BLOCK

DATA_BLOCK "GA2_1_AI_2"	// DB 34
VERSION : 0.1
  STRUCT
   B_0 : BYTE ;
   B_1 : BYTE ;
   B_2 : BYTE ;
   B_3 : BYTE ;
   B_4 : BYTE ;
   B_5 : BYTE ;
   B_6 : BYTE ;
   B_7 : BYTE ;
   B_8 : BYTE ;
   B_9 : BYTE ;
   B_10 : BYTE ;
   B_11 : BYTE ;
   B_12 : BYTE ;
   B_13 : BYTE ;
   B_14 : BYTE ;
   B_15 : BYTE ;
   B_16 : BYTE ;
  END_STRUCT ;	
BEGIN
END_DATA_BLOCK

DATA_BLOCK "KD1_1_AI"	// DB 35
VERSION : 0.1
  STRUCT
   B_0 : BYTE ;
   B_1 : BYTE ;
   B_2 : BYTE ;
   B_3 : BYTE ;
   B_4 : BYTE ;
   B_5 : BYTE ;
   B_6 : BYTE ;
   B_7 : BYTE ;
   B_8 : BYTE ;
   B_9 : BYTE ;
   B_10 : BYTE ;
   B_11 : BYTE ;
   B_12 : BYTE ;
  END_STRUCT ;	
BEGIN
END_DATA_BLOCK

DATA_BLOCK "GA2_2_AI_1"	// DB 36
VERSION : 0.1
  STRUCT
   B_0 : BYTE ;
   B_1 : BYTE ;
   B_2 : BYTE ;
   B_3 : BYTE ;
   B_4 : BYTE ;
   B_5 : BYTE ;
   B_6 : BYTE ;
   B_7 : BYTE ;
   B_8 : BYTE ;
   B_9 : BYTE ;
   B_10 : BYTE ;
   B_11 : BYTE ;
   B_12 : BYTE ;
   B_13 : BYTE ;
   B_14 : BYTE ;
   B_15 : BYTE ;
   B_16 : BYTE ;
   B_17 : BYTE ;
   B_18 : BYTE ;
   B_19 : BYTE ;
   B_20 : BYTE ;
  END_STRUCT ;	
BEGIN
END_DATA_BLOCK

DATA_BLOCK "GA2_2_AI_2"	// DB 37
VERSION : 0.1
  STRUCT
   B_0 : BYTE ;
   B_1 : BYTE ;
   B_2 : BYTE ;
   B_3 : BYTE ;
   B_4 : BYTE ;
   B_5 : BYTE ;
   B_6 : BYTE ;
   B_7 : BYTE ;
   B_8 : BYTE ;
   B_9 : BYTE ;
   B_10 : BYTE ;
   B_11 : BYTE ;
   B_12 : BYTE ;
   B_13 : BYTE ;
   B_14 : BYTE ;
   B_15 : BYTE ;
   B_16 : BYTE ;
  END_STRUCT ;	
BEGIN
END_DATA_BLOCK

DATA_BLOCK "KD1_1_AI_2"	// DB 38
VERSION : 0.1
  STRUCT
   B_0 : BYTE ;
   B_1 : BYTE ;
   B_2 : BYTE ;
   B_3 : BYTE ;
   B_4 : BYTE ;
   B_5 : BYTE ;
   B_6 : BYTE ;
   B_7 : BYTE ;
   B_8 : BYTE ;
   B_9 : BYTE ;
   B_10 : BYTE ;
   B_11 : BYTE ;
   B_12 : BYTE ;
   B_13 : BYTE ;
   B_14 : BYTE ;
   B_15 : BYTE ;
   B_16 : BYTE ;
   B_17 : BYTE ;
   B_18 : BYTE ;
   B_19 : BYTE ;
   B_20 : BYTE ;
   B_21 : BYTE ;
   B_22 : BYTE ;
   B_23 : BYTE ;
   B_24 : BYTE ;
   B_25 : BYTE ;
   B_26 : BYTE ;
   B_27 : BYTE ;
   B_28 : BYTE ;
   B_29 : BYTE ;
   B_30 : BYTE ;
   B_31 : BYTE ;
   B_32 : BYTE ;
   B_33 : BYTE ;
   B_34 : BYTE ;
   B_35 : BYTE ;
   B_36 : BYTE ;
   B_37 : BYTE ;
   B_38 : BYTE ;
   B_39 : BYTE ;
   B_40 : BYTE ;
  END_STRUCT ;	
BEGIN
END_DATA_BLOCK

DATA_BLOCK "KD1_1_AI_3"	// DB 39
VERSION : 0.1
  STRUCT
   B_0 : BYTE ;
   B_1 : BYTE ;
   B_2 : BYTE ;
   B_3 : BYTE ;
   B_4 : BYTE ;
   B_5 : BYTE ;
   B_6 : BYTE ;
   B_7 : BYTE ;
   B_8 : BYTE ;
   B_9 : BYTE ;
   B_10 : BYTE ;
   B_11 : BYTE ;
   B_12 : BYTE ;
   B_13 : BYTE ;
   B_14 : BYTE ;
   B_15 : BYTE ;
   B_16 : BYTE ;
   B_17 : BYTE ;
   B_18 : BYTE ;
   B_19 : BYTE ;
   B_20 : BYTE ;
   B_21 : BYTE ;
   B_22 : BYTE ;
   B_23 : BYTE ;
   B_24 : BYTE ;
   B_25 : BYTE ;
   B_26 : BYTE ;
   B_27 : BYTE ;
   B_28 : BYTE ;
   B_29 : BYTE ;
   B_30 : BYTE ;
   B_31 : BYTE ;
   B_32 : BYTE ;
  END_STRUCT ;	
BEGIN
END_DATA_BLOCK

DATA_BLOCK "KD1_1_AI_4"	// DB 40
VERSION : 0.1
  STRUCT
   B_0 : BYTE ;
   B_1 : BYTE ;
   B_2 : BYTE ;
   B_3 : BYTE ;
   B_4 : BYTE ;
   B_5 : BYTE ;
   B_6 : BYTE ;
   B_7 : BYTE ;
   B_8 : BYTE ;
   B_9 : BYTE ;
   B_10 : BYTE ;
   B_11 : BYTE ;
   B_12 : BYTE ;
   B_13 : BYTE ;
   B_14 : BYTE ;
   B_15 : BYTE ;
   B_16 : BYTE ;
   B_17 : BYTE ;
   B_18 : BYTE ;
   B_19 : BYTE ;
   B_20 : BYTE ;
   B_21 : BYTE ;
   B_22 : BYTE ;
   B_23 : BYTE ;
   B_24 : BYTE ;
   B_25 : BYTE ;
   B_26 : BYTE ;
   B_27 : BYTE ;
   B_28 : BYTE ;
   B_29 : BYTE ;
   B_30 : BYTE ;
   B_31 : BYTE ;
   B_32 : BYTE ;
  END_STRUCT ;	
BEGIN
END_DATA_BLOCK

DATA_BLOCK "KD1_1_AI_5"	// DB 41
VERSION : 0.1
  STRUCT
   B_0 : BYTE ;
   B_1 : BYTE ;
   B_2 : BYTE ;
   B_3 : BYTE ;
   B_4 : BYTE ;
   B_5 : BYTE ;
   B_6 : BYTE ;
   B_7 : BYTE ;
   B_8 : BYTE ;
   B_9 : BYTE ;
   B_10 : BYTE ;
   B_11 : BYTE ;
   B_12 : BYTE ;
  END_STRUCT ;	
BEGIN
END_DATA_BLOCK

DATA_BLOCK "KD1_1_Coils"	// DB 42
VERSION : 0.1
  STRUCT
   B_0 : BYTE ;
   B_1 : BYTE ;
   Running_Stopped : BOOL ;
   Load_Unload : BOOL ;
   General_Warning : BOOL ;
   GeneralShutdownWarning : BOOL ;
   GeneralShutdown : BOOL ;
   GeneralService : BOOL ;
   GeneralStartFailure : BOOL ;
   EmergencyStop : BOOL ;
   Automatic_Manual : BOOL ;
   Remote_Local : BOOL ;
   DB_VAR : INT ;	//Temporary placeholder variable
  END_STRUCT ;	
BEGIN
END_DATA_BLOCK

DATA_BLOCK "BD1_ARR_AI"	// DB 43
VERSION : 0.1
  STRUCT
   arBytes : ARRAY  [1 .. 50 ] OF BYTE ;
  END_STRUCT ;	
BEGIN
END_DATA_BLOCK

DATA_BLOCK "BD_AI_2"	// DB 44
VERSION : 0.1
  STRUCT
   B_0 : BYTE ;
   B_1 : BYTE ;
   B_2 : BYTE ;
   B_3 : BYTE ;
   B_4 : BYTE ;
   B_5 : BYTE ;
   B_6 : BYTE ;
   B_7 : BYTE ;
   B_8 : BYTE ;
   B_9 : BYTE ;
   B_10 : BYTE ;
   B_11 : BYTE ;
   B_12 : BYTE ;
  END_STRUCT ;	
BEGIN
END_DATA_BLOCK

DATA_BLOCK "BD_AI_3"	// DB 45
VERSION : 0.1
  STRUCT
   B_0 : BYTE ;
   B_1 : BYTE ;
   B_2 : BYTE ;
   B_3 : BYTE ;
  END_STRUCT ;	
BEGIN
END_DATA_BLOCK

DATA_BLOCK "BD_DO_1"	// DB 46
VERSION : 0.1
  STRUCT
   arBytes : ARRAY  [0 .. 5 ] OF BYTE ;
  END_STRUCT ;	
BEGIN
END_DATA_BLOCK

DATA_BLOCK "BD_DO_2"	// DB 47
VERSION : 0.1
  STRUCT
   arBytes : ARRAY  [0 .. 13 ] OF BYTE ;
  END_STRUCT ;	
BEGIN
END_DATA_BLOCK

DATA_BLOCK "GA1_1_DO"	// DB 48
VERSION : 0.1
  STRUCT
   arBytes : ARRAY  [0 .. 14 ] OF BYTE ;
  END_STRUCT ;	
BEGIN
END_DATA_BLOCK

DATA_BLOCK "GA1_2_DO"	// DB 49
VERSION : 0.1
  STRUCT
   arBytes : ARRAY  [0 .. 14 ] OF BYTE ;
  END_STRUCT ;	
BEGIN
END_DATA_BLOCK

DATA_BLOCK "GA2_1_DO"	// DB 50
VERSION : 0.1
  STRUCT
   arBytes : ARRAY  [0 .. 14 ] OF BYTE ;
  END_STRUCT ;	
BEGIN
END_DATA_BLOCK

DATA_BLOCK "GA2_2_DO"	// DB 51
VERSION : 0.1
  STRUCT
   arBytes : ARRAY  [0 .. 14 ] OF BYTE ;
  END_STRUCT ;	
BEGIN
END_DATA_BLOCK

DATA_BLOCK "BD_REAL"	// DB 52
VERSION : 0.1
  STRUCT
   PressureVesselA : REAL ;
   PressureVesselB : REAL ;
   InletDryer : REAL ;
   HeaterOut : REAL ;
   RegenerationAirOutlet : REAL ;
   DryerPressureDewpoint : REAL ;
  END_STRUCT ;	
BEGIN
END_DATA_BLOCK

DATA_BLOCK "KB1_1_REAL"	// DB 53
VERSION : 0.1
  STRUCT
   InputPressure : REAL ;
   PressureChangeOnFiltr : REAL ;
   OilPressure : REAL ;
   PromCoolerPressure : REAL ;
   TafterCompressor : REAL ;
   TafterStep_1 : REAL ;
   TafterStep_2 : REAL ;
   TafterStep_3 : REAL ;
   TinputCoolWater : REAL ;
   TwaterAfterStepND : REAL ;
   ToutCoolWater : REAL ;
   Toil : REAL ;
   Tmotor_U1 : REAL ;
   Tmotor_V1 : REAL ;
   Tmotor_W1 : REAL ;
  END_STRUCT ;	
BEGIN
END_DATA_BLOCK

DATA_BLOCK "KB1_2_REAL"	// DB 54
VERSION : 0.1
  STRUCT
   InputPressure : REAL ;
   PressureChangeOnFiltr : REAL ;
   OilPressure : REAL ;
   PromCoolerPressure : REAL ;
   TafterCompressor : REAL ;
   TafterStep_1 : REAL ;
   TafterStep_2 : REAL ;
   TafterStep_3 : REAL ;
   TinputCoolWater : REAL ;
   TwaterAfterStepND : REAL ;
   ToutCoolWater : REAL ;
   Toil : REAL ;
   Tmotor_U1 : REAL ;
   Tmotor_V1 : REAL ;
   Tmotor_W1 : REAL ;
  END_STRUCT ;	
BEGIN
END_DATA_BLOCK

DATA_BLOCK "KB2_REAL"	// DB 55
VERSION : 0.1
  STRUCT
   OilPressureReductor : REAL ;
   PressureChangeOnFiltr : REAL ;
   PressureChangeOnOilFiltr : REAL ;
   Step3OutPressure : REAL ;
   ToilReductor : REAL ;
   TinputCoolWater : REAL ;
   TinputStep_2 : REAL ;
   TinputStep_3 : REAL ;
   TafterCompressor : REAL ;
   ToilTank : REAL ;
   Tmotor_U1 : REAL ;
   Tmotor_V1 : REAL ;
   Tmotor_W1 : REAL ;
   OutPressure : REAL ;
   Aject2Step : REAL ;
   PchangeStep2 : REAL ;
   TmotorBearier_D_End : REAL ;
   TmotorBearier_ND_End : REAL ;
   Vibration_1 : REAL ;
   Vibration_2 : REAL ;
   Vibration_3 : REAL ;
  END_STRUCT ;	
BEGIN
END_DATA_BLOCK

DATA_BLOCK "PO1_1_REAL"	// DB 56
VERSION : 0.1
  STRUCT
   CondPressure : REAL ;
   EvaporatingPressureComp : REAL ;
   EvaporatingPressureHE_1 : REAL ;
   EvaporatingPressureHE_2 : REAL ;
   Dewpoint_1 : REAL ;
   Freon_1 : REAL ;
   Dewpoint_2 : REAL ;
   Freon_11 : REAL ;
   ToutAir : REAL ;
   TfreonIn : REAL ;
   TfreonOut : REAL ;
  END_STRUCT ;	
BEGIN
END_DATA_BLOCK

DATA_BLOCK "PO1_2_REAL"	// DB 57
VERSION : 0.1
  STRUCT
   CondPressure : REAL ;
   EvaporatingPressureComp : REAL ;
   EvaporatingPressureHE_1 : REAL ;
   EvaporatingPressureHE_2 : REAL ;
   Dewpoint_1 : REAL ;
   Freon_1 : REAL ;
   Dewpoint_2 : REAL ;
   Freon_11 : REAL ;
   ToutAir : REAL ;
   TfreonIn : REAL ;
   TfreonOut : REAL ;
  END_STRUCT ;	
BEGIN
END_DATA_BLOCK

DATA_BLOCK "GA1_1_REAL"	// DB 58
VERSION : 0.1
  STRUCT
   AirGeneratorIn : REAL ;
   PressureVesselA : REAL ;
   PressureVesselB : REAL ;
   NitrogenOutlet : REAL ;
   AirGeneratorIn1 : REAL ;
   DryerPressureDewpoint : REAL ;
   NitrogenDewpoint : REAL ;
   OutletFlow : REAL ;
   OxygenPurity : REAL ;
  END_STRUCT ;	
BEGIN
END_DATA_BLOCK

DATA_BLOCK "GA1_2_REAL"	// DB 59
VERSION : 0.1
  STRUCT
   AirGeneratorIn : REAL ;
   PressureVesselA : REAL ;
   PressureVesselB : REAL ;
   NitrogenOutlet : REAL ;
   AirGeneratorIn1 : REAL ;
   DryerPressureDewpoint : REAL ;
   NitrogenDewpoint : REAL ;
   OutletFlow : REAL ;
   OxygenPurity : REAL ;
  END_STRUCT ;	
BEGIN
END_DATA_BLOCK

DATA_BLOCK "GA2_1_REAL"	// DB 60
VERSION : 0.1
  STRUCT
   AirGeneratorIn : REAL ;
   PressureVesselA : REAL ;
   PressureVesselB : REAL ;
   NitrogenOutlet : REAL ;
   AirGeneratorIn1 : REAL ;
   DryerPressureDewpoint : REAL ;
   NitrogenDewpoint : REAL ;
   OutletFlow : REAL ;
   OxygenPurity : REAL ;
  END_STRUCT ;	
BEGIN
END_DATA_BLOCK

DATA_BLOCK "GA2_2_REAL"	// DB 61
VERSION : 0.1
  STRUCT
   AirGeneratorIn : REAL ;
   PressureVesselA : REAL ;
   PressureVesselB : REAL ;
   NitrogenOutlet : REAL ;
   AirGeneratorIn1 : REAL ;
   DryerPressureDewpoint : REAL ;
   NitrogenDewpoint : REAL ;
   OutletFlow : REAL ;
   OxygenPurity : REAL ;
  END_STRUCT ;	
BEGIN
END_DATA_BLOCK

DATA_BLOCK "KD_REAL"	// DB 62
VERSION : 0.1
  STRUCT
   CompressorOutlet : REAL ;
   OilPressure : REAL ;
   Element_1_Inlet : REAL ;
   Element_1A_Outlet : REAL ;
   Element_2A_Outlet : REAL ;
   Element_1B_Outlet : REAL ;
   Element_2B_Outlet : REAL ;
   CoolingWaterInT : REAL ;
   CoolingWaterOut : REAL ;
   OilTemperature : REAL ;
   SuctionTemperature : REAL ;
   MotorWinding1U1 : REAL ;
   MotorWinding1V1 : REAL ;
   MotorWinding1W1 : REAL ;
   RodDrop1 : REAL ;
   RodDrop2 : REAL ;
   NitrogenDewpoint : REAL ;
   RodDrop3 : REAL ;
   RodDrop4 : REAL ;
  END_STRUCT ;	
BEGIN
END_DATA_BLOCK

DATA_BLOCK "ModbusVars"	// DB 63
VERSION : 0.1
  STRUCT
   wCync : WORD ;
  END_STRUCT ;	
BEGIN
END_DATA_BLOCK

DATA_BLOCK "BD_Outputs_1"	// DB 64
VERSION : 0.1
  STRUCT
   DryerMotor : WORD ;
   PDPAlarm : WORD ;
   GeneralShutdown : WORD ;
   GeneralWarning : WORD ;
   LowPressureAlarm : WORD ;
  END_STRUCT ;	
BEGIN
END_DATA_BLOCK

DATA_BLOCK "BD_Outputs_2"	// DB 65
VERSION : 0.1
  STRUCT
   BlowerContactor : WORD ;
   MainHeaters : WORD ;
   RegulatingHeaters : WORD ;
   ValveV1Opened : WORD ;
   ValveV1Closed : WORD ;
   ValveV2Opened : WORD ;
   ValveV2Closed : WORD ;
   RegValveVesselA : WORD ;
   RegValveVesselB : WORD ;
   CoolingAirValveAOpen : WORD ;
   CoolingAirValveBOpen : WORD ;
   PressureReliefValveA : WORD ;
   PressureReliefValvegB : WORD ;
  END_STRUCT ;	
BEGIN
END_DATA_BLOCK

DATA_BLOCK "PO1_1_Outputs"	// DB 66
VERSION : 0.1
  STRUCT
   EEV1 : REAL ;
   EEV2 : REAL ;
   HGBP1 : REAL ;
   HGBP2 : REAL ;
  END_STRUCT ;	
BEGIN
END_DATA_BLOCK

DATA_BLOCK "PO1_2_Outputs"	// DB 67
VERSION : 0.1
  STRUCT
   EEV1 : REAL ;
   EEV2 : REAL ;
   HGBP1 : REAL ;
   HGBP2 : REAL ;
  END_STRUCT ;	
BEGIN
END_DATA_BLOCK

DATA_BLOCK "GA1_1_Outputs"	// DB 68
VERSION : 0.1
  STRUCT
   InletValveVesselA : WORD ;
   InletValveVesselB : WORD ;
   EqualizationValve : WORD ;
   RegenValveVesselA : WORD ;
   RegenValveVesselB : WORD ;
   ProductionValveVesselA : WORD ;
   ProductionValveVesselB : WORD ;
   SolenoidValves : WORD ;
   ConsumerValve : WORD ;
   InletFlushingValve : WORD ;
   ExhaustValve : WORD ;
   Running : WORD ;
   SecondRunning : WORD ;
   GeneralWarning : WORD ;
   GeneralShutdown : WORD ;
  END_STRUCT ;	
BEGIN
END_DATA_BLOCK

DATA_BLOCK "GA1_2_Outputs"	// DB 69
VERSION : 0.1
  STRUCT
   InletValveVesselA : WORD ;
   InletValveVesselB : WORD ;
   EqualizationValve : WORD ;
   RegenValveVesselA : WORD ;
   RegenValveVesselB : WORD ;
   ProductionValveVesselA : WORD ;
   ProductionValveVesselB : WORD ;
   SolenoidValves : WORD ;
   ConsumerValve : WORD ;
   InletFlushingValve : WORD ;
   ExhaustValve : WORD ;
   Running : WORD ;
   SecondRunning : WORD ;
   GeneralWarning : WORD ;
   GeneralShutdown : WORD ;
  END_STRUCT ;	
BEGIN
END_DATA_BLOCK

DATA_BLOCK DB 70
AUTHOR : T.HAJNAL
FAMILY : MODBUS
VERSION : 0.0
"MBMAREQ"
BEGIN
END_DATA_BLOCK

DATA_BLOCK DB 71
AUTHOR : T.HAJNAL
FAMILY : MODBUS
VERSION : 0.0
"MBMAREQ"
BEGIN
END_DATA_BLOCK

DATA_BLOCK DB 72
AUTHOR : T.HAJNAL
FAMILY : MODBUS
VERSION : 0.0
"MBMAREQ"
BEGIN
END_DATA_BLOCK

DATA_BLOCK DB 73
AUTHOR : T.HAJNAL
FAMILY : MODBUS
VERSION : 0.0
"MBMAREQ"
BEGIN
END_DATA_BLOCK

DATA_BLOCK DB 74
AUTHOR : T.HAJNAL
FAMILY : MODBUS
VERSION : 0.0
"MBMAREQ"
BEGIN
END_DATA_BLOCK

DATA_BLOCK DB 75
AUTHOR : T.HAJNAL
FAMILY : MODBUS
VERSION : 0.0
"MBMAREQ"
BEGIN
END_DATA_BLOCK

DATA_BLOCK DB 76
AUTHOR : T.HAJNAL
FAMILY : MODBUS
VERSION : 0.0
"MBMAREQ"
BEGIN
END_DATA_BLOCK

DATA_BLOCK DB 77
AUTHOR : T.HAJNAL
FAMILY : MODBUS
VERSION : 0.0
"MBMAREQ"
BEGIN
END_DATA_BLOCK

DATA_BLOCK DB 78
AUTHOR : T.HAJNAL
FAMILY : MODBUS
VERSION : 0.0
"MBMAREQ"
BEGIN
END_DATA_BLOCK

DATA_BLOCK DB 79
AUTHOR : T.HAJNAL
FAMILY : MODBUS
VERSION : 0.0
"MBMAREQ"
BEGIN
END_DATA_BLOCK

DATA_BLOCK DB 80
AUTHOR : T.HAJNAL
FAMILY : MODBUS
VERSION : 0.0
"MBMAREQ"
BEGIN
END_DATA_BLOCK

DATA_BLOCK DB 81
AUTHOR : T.HAJNAL
FAMILY : MODBUS
VERSION : 0.0
"MBMAREQ"
BEGIN
END_DATA_BLOCK

DATA_BLOCK DB 82
AUTHOR : T.HAJNAL
FAMILY : MODBUS
VERSION : 0.0
"MBMAREQ"
BEGIN
END_DATA_BLOCK

DATA_BLOCK DB 83
AUTHOR : T.HAJNAL
FAMILY : MODBUS
VERSION : 0.0
"MBMAREQ"
BEGIN
END_DATA_BLOCK

DATA_BLOCK DB 84
AUTHOR : T.HAJNAL
FAMILY : MODBUS
VERSION : 0.0
"MBMAREQ"
BEGIN
END_DATA_BLOCK

DATA_BLOCK DB 85
AUTHOR : T.HAJNAL
FAMILY : MODBUS
VERSION : 0.0
"MBMAREQ"
BEGIN
END_DATA_BLOCK

DATA_BLOCK DB 86
AUTHOR : T.HAJNAL
FAMILY : MODBUS
VERSION : 0.0
"MBMAREQ"
BEGIN
END_DATA_BLOCK

DATA_BLOCK DB 87
AUTHOR : T.HAJNAL
FAMILY : MODBUS
VERSION : 0.0
"MBMAREQ"
BEGIN
END_DATA_BLOCK

DATA_BLOCK DB 88
AUTHOR : T.HAJNAL
FAMILY : MODBUS
VERSION : 0.0
"MBMAREQ"
BEGIN
END_DATA_BLOCK

DATA_BLOCK DB 89
AUTHOR : T.HAJNAL
FAMILY : MODBUS
VERSION : 0.0
"MBMAREQ"
BEGIN
END_DATA_BLOCK

DATA_BLOCK DB 90
AUTHOR : T.HAJNAL
FAMILY : MODBUS
VERSION : 0.0
"MBMAREQ"
BEGIN
END_DATA_BLOCK

DATA_BLOCK DB 91
AUTHOR : T.HAJNAL
FAMILY : MODBUS
VERSION : 0.0
"MBMAREQ"
BEGIN
END_DATA_BLOCK

DATA_BLOCK DB 92
AUTHOR : T.HAJNAL
FAMILY : MODBUS
VERSION : 0.0
"MBMAREQ"
BEGIN
END_DATA_BLOCK

DATA_BLOCK DB 93
AUTHOR : T.HAJNAL
FAMILY : MODBUS
VERSION : 0.0
"MBMAREQ"
BEGIN
END_DATA_BLOCK

DATA_BLOCK DB 94
AUTHOR : T.HAJNAL
FAMILY : MODBUS
VERSION : 0.0
"MBMAREQ"
BEGIN
END_DATA_BLOCK

DATA_BLOCK DB 95
AUTHOR : T.HAJNAL
FAMILY : MODBUS
VERSION : 0.0
"MBMAREQ"
BEGIN
END_DATA_BLOCK

DATA_BLOCK DB 96
AUTHOR : T.HAJNAL
FAMILY : MODBUS
VERSION : 0.0
"MBMAREQ"
BEGIN
END_DATA_BLOCK

DATA_BLOCK "GA2_1_Outputs"	// DB 97
VERSION : 0.1
  STRUCT
   InletValveVesselA : WORD ;
   InletValveVesselB : WORD ;
   EqualizationValve : WORD ;
   RegenValveVesselA : WORD ;
   RegenValveVesselB : WORD ;
   ProductionValveVesselA : WORD ;
   ProductionValveVesselB : WORD ;
   SolenoidValves : WORD ;
   ConsumerValve : WORD ;
   InletFlushingValve : WORD ;
   ExhaustValve : WORD ;
   Running : WORD ;
   SecondRunning : WORD ;
   GeneralWarning : WORD ;
   GeneralShutdown : WORD ;
  END_STRUCT ;	
BEGIN
END_DATA_BLOCK

DATA_BLOCK "GA2_2_Outputs"	// DB 98
VERSION : 0.1
  STRUCT
   InletValveVesselA : WORD ;
   InletValveVesselB : WORD ;
   EqualizationValve : WORD ;
   RegenValveVesselA : WORD ;
   RegenValveVesselB : WORD ;
   ProductionValveVesselA : WORD ;
   ProductionValveVesselB : WORD ;
   SolenoidValves : WORD ;
   ConsumerValve : WORD ;
   InletFlushingValve : WORD ;
   ExhaustValve : WORD ;
   Running : WORD ;
   SecondRunning : WORD ;
   GeneralWarning : WORD ;
   GeneralShutdown : WORD ;
  END_STRUCT ;	
BEGIN
END_DATA_BLOCK

DATA_BLOCK "BD_OutputBytes_1"	// DB 99
VERSION : 0.1
  STRUCT
   arBytes : ARRAY  [0 .. 9 ] OF BYTE ;
  END_STRUCT ;	
BEGIN
END_DATA_BLOCK

DATA_BLOCK DB 100
AUTHOR : T.HAJNAL
FAMILY : MODBUS
VERSION : 0.0
"MBMAREQ"
BEGIN
END_DATA_BLOCK

DATA_BLOCK DB 101
AUTHOR : T.HAJNAL
FAMILY : MODBUS
VERSION : 0.0
"MBMAREQ"
BEGIN
END_DATA_BLOCK

DATA_BLOCK DB 102
AUTHOR : T.HAJNAL
FAMILY : MODBUS
VERSION : 0.0
"MBMAREQ"
BEGIN
END_DATA_BLOCK

DATA_BLOCK DB 103
AUTHOR : T.HAJNAL
FAMILY : MODBUS
VERSION : 0.0
"MBMAREQ"
BEGIN
END_DATA_BLOCK

DATA_BLOCK DB 104
AUTHOR : T.HAJNAL
FAMILY : MODBUS
VERSION : 0.0
"MBMAREQ"
BEGIN
END_DATA_BLOCK

DATA_BLOCK DB 105
AUTHOR : T.HAJNAL
FAMILY : MODBUS
VERSION : 0.0
"MBMAREQ"
BEGIN
END_DATA_BLOCK

DATA_BLOCK DB 106
AUTHOR : T.HAJNAL
FAMILY : MODBUS
VERSION : 0.0
"MBMAREQ"
BEGIN
END_DATA_BLOCK

DATA_BLOCK DB 107
AUTHOR : T.HAJNAL
FAMILY : MODBUS
VERSION : 0.0
"MBMAREQ"
BEGIN
END_DATA_BLOCK

DATA_BLOCK DB 108
AUTHOR : T.HAJNAL
FAMILY : MODBUS
VERSION : 0.0
"MBMAREQ"
BEGIN
END_DATA_BLOCK

DATA_BLOCK DB 109
AUTHOR : T.HAJNAL
FAMILY : MODBUS
VERSION : 0.0
"MBMAREQ"
BEGIN
END_DATA_BLOCK

DATA_BLOCK DB 110
AUTHOR : T.HAJNAL
FAMILY : MODBUS
VERSION : 0.0
"MBMAREQ"
BEGIN
END_DATA_BLOCK

DATA_BLOCK "BD_OutputBytes_2"	// DB 111
VERSION : 0.1
  STRUCT
   arBytes : ARRAY  [0 .. 25 ] OF BYTE ;
  END_STRUCT ;	
BEGIN
END_DATA_BLOCK

DATA_BLOCK "PO1_1_OutBytes"	// DB 112
VERSION : 0.1
  STRUCT
   arBytes : ARRAY  [0 .. 7 ] OF BYTE ;
  END_STRUCT ;	
BEGIN
END_DATA_BLOCK

DATA_BLOCK "PO1_2_OutBytes"	// DB 113
VERSION : 0.1
  STRUCT
   arBytes : ARRAY  [0 .. 7 ] OF BYTE ;
  END_STRUCT ;	
BEGIN
END_DATA_BLOCK

DATA_BLOCK "GA1_1_OutBytes"	// DB 114
VERSION : 0.1
  STRUCT
   arBytes : ARRAY  [0 .. 29 ] OF BYTE ;
  END_STRUCT ;	
BEGIN
END_DATA_BLOCK

DATA_BLOCK "GA1_2_OutBytes"	// DB 115
VERSION : 0.1
  STRUCT
   arBytes : ARRAY  [0 .. 29 ] OF BYTE ;
  END_STRUCT ;	
BEGIN
END_DATA_BLOCK

DATA_BLOCK "GA2_1_OutBytes"	// DB 116
VERSION : 0.1
  STRUCT
   arBytes : ARRAY  [0 .. 29 ] OF BYTE ;
  END_STRUCT ;	
BEGIN
END_DATA_BLOCK

DATA_BLOCK "GA2_2_OutBytes"	// DB 117
VERSION : 0.1
  STRUCT
   arBytes : ARRAY  [0 .. 29 ] OF BYTE ;
  END_STRUCT ;	
BEGIN
END_DATA_BLOCK

DATA_BLOCK "StartStop"	// DB 118
VERSION : 0.1
  STRUCT
   xBD_Start : BOOL ;
   xBD_Stop : BOOL ;
   xKB1_1_Start : BOOL ;
   xKB1_1_Stop : BOOL ;
   xKB1_2_Start : BOOL ;
   xKB1_2_Stop : BOOL ;
   xKB2_Start : BOOL ;
   xKB2_Stop : BOOL ;
   xPO1_1_Start : BOOL ;
   xPO1_1_Stop : BOOL ;
   xPO1_2_Start : BOOL ;
   xPO1_2_Stop : BOOL ;
   xGA1_1_Start : BOOL ;
   xGA1_1_Stop : BOOL ;
   xGA1_2_Start : BOOL ;
   xGA1_2_Stop : BOOL ;
   xGA2_1_Start : BOOL ;
   xGA2_1_Stop : BOOL ;
   xGA2_2_Start : BOOL ;
   xGA2_2_Stop : BOOL ;
   xKD_Start : BOOL ;
   xKD_Stop : BOOL ;
   xPO2_Start : BOOL ;
   xPO2_Stop : BOOL ;
  END_STRUCT ;	
BEGIN
END_DATA_BLOCK

DATA_BLOCK "StartStopBytes"	// DB 119
VERSION : 0.1
  STRUCT
   BD_High : BYTE ;
   BD_StartStop : BYTE ;
   KB1_1_High : BYTE ;
   KB1_1_StartStop : BYTE ;
   KB1_2_High : BYTE ;
   KB1_2_StartStop : BYTE ;
   KB2_High : BYTE ;
   KB2_StartStop : BYTE ;
   PO1_1_High : BYTE ;
   PO1_1_StartStop : BYTE ;
   PO1_2_High : BYTE ;
   PO1_2_StartStop : BYTE ;
   GA1_1_High : BYTE ;
   GA1_1_StartStop : BYTE ;
   GA1_2_High : BYTE ;
   GA1_2_StartStop : BYTE ;
   GA2_1_High : BYTE ;
   GA2_1_StartStop : BYTE ;
   GA2_2_High : BYTE ;
   GA2_2_StartStop : BYTE ;
   KD_High : BYTE ;
   KD_StartStop : BYTE ;
   PO2_High : BYTE ;
   PO2_StartStop : BYTE ;
  END_STRUCT ;	
BEGIN
END_DATA_BLOCK

DATA_BLOCK DB 120
AUTHOR : T.HAJNAL
FAMILY : MODBUS
VERSION : 0.0
"MBMAREQ"
BEGIN
END_DATA_BLOCK

DATA_BLOCK DB 121
AUTHOR : T.HAJNAL
FAMILY : MODBUS
VERSION : 0.0
"MBMAREQ"
BEGIN
END_DATA_BLOCK

DATA_BLOCK DB 122
AUTHOR : T.HAJNAL
FAMILY : MODBUS
VERSION : 0.0
"MBMAREQ"
BEGIN
END_DATA_BLOCK

DATA_BLOCK DB 123
AUTHOR : T.HAJNAL
FAMILY : MODBUS
VERSION : 0.0
"MBMAREQ"
BEGIN
END_DATA_BLOCK

DATA_BLOCK DB 124
AUTHOR : T.HAJNAL
FAMILY : MODBUS
VERSION : 0.0
"MBMAREQ"
BEGIN
END_DATA_BLOCK

DATA_BLOCK DB 125
AUTHOR : T.HAJNAL
FAMILY : MODBUS
VERSION : 0.0
"MBMAREQ"
BEGIN
END_DATA_BLOCK

DATA_BLOCK DB 126
AUTHOR : T.HAJNAL
FAMILY : MODBUS
VERSION : 0.0
"MBMAREQ"
BEGIN
END_DATA_BLOCK

DATA_BLOCK DB 127
AUTHOR : T.HAJNAL
FAMILY : MODBUS
VERSION : 0.0
"MBMAREQ"
BEGIN
END_DATA_BLOCK

DATA_BLOCK "KB2_AI_Bearer"	// DB 128
VERSION : 0.1
  STRUCT
   B_0 : BYTE ;
   B_1 : BYTE ;
   B_2 : BYTE ;
   B_3 : BYTE ;
   B_4 : BYTE ;
   B_5 : BYTE ;
   B_6 : BYTE ;
   B_7 : BYTE ;
   B_8 : BYTE ;
  END_STRUCT ;	
BEGIN
END_DATA_BLOCK

DATA_BLOCK "KB2_AI_Vibration"	// DB 129
VERSION : 0.1
  STRUCT
   B_0 : BYTE ;
   B_1 : BYTE ;
   B_2 : BYTE ;
   B_3 : BYTE ;
   B_4 : BYTE ;
   B_5 : BYTE ;
   B_6 : BYTE ;
   B_7 : BYTE ;
   B_8 : BYTE ;
   B_9 : BYTE ;
   B_10 : BYTE ;
   B_11 : BYTE ;
   B_12 : BYTE ;
  END_STRUCT ;	
BEGIN
END_DATA_BLOCK

DATA_BLOCK "ModbusAddresses"	// DB 130
VERSION : 0.1
  STRUCT
   BD_Addr : INT  := 10;	//Temporary placeholder variable
   KB1_1_Addr : INT  := 3;
   KB1_2_Addr : INT  := 4;
   KB2_Addr : INT  := 5;
   PO1_1_Addr : INT  := 6;
   PO1_2_Addr : INT  := 7;
   GA1_1_Addr : INT  := 11;
   GA1_2_Addr : INT  := 12;
   GA2_1_Addr : INT  := 14;
   GA2_2_Addr : INT  := 13;
   KD1_Addr : INT  := 15;
   PO2_Addr : INT  := 9;
  END_STRUCT ;	
BEGIN
   BD_Addr := 10;
   KB1_1_Addr := 3;
   KB1_2_Addr := 4;
   KB2_Addr := 5;
   PO1_1_Addr := 6;
   PO1_2_Addr := 7;
   GA1_1_Addr := 11;
   GA1_2_Addr := 12;
   GA2_1_Addr := 14;
   GA2_2_Addr := 13;
   KD1_Addr := 15;
   PO2_Addr := 9;
END_DATA_BLOCK

DATA_BLOCK "PO2_AI"	// DB 131
VERSION : 0.1
  STRUCT
   B_0 : BYTE ;
   B_1 : BYTE ;
   B_2 : BYTE ;
   B_3 : BYTE ;
   B_4 : BYTE ;
   B_5 : BYTE ;
   B_6 : BYTE ;
   B_7 : BYTE ;
   B_8 : BYTE ;
   B_9 : BYTE ;
   B_10 : BYTE ;
   B_11 : BYTE ;
   B_12 : BYTE ;
   B_13 : BYTE ;
   B_14 : BYTE ;
   B_15 : BYTE ;
   B_16 : BYTE ;
   B_17 : BYTE ;
   B_18 : BYTE ;
   B_19 : BYTE ;
   B_20 : BYTE ;
   B_21 : BYTE ;
   B_22 : BYTE ;
   B_23 : BYTE ;
   B_24 : BYTE ;
   B_25 : BYTE ;
   B_26 : BYTE ;
   B_27 : BYTE ;
   B_28 : BYTE ;
  END_STRUCT ;	
BEGIN
END_DATA_BLOCK

DATA_BLOCK "PO2_Reals"	// DB 132
VERSION : 0.1
  STRUCT
   T_Dryer_1 : REAL ;
   T_Dryer_2 : REAL ;
   T_Dryer_3 : REAL ;
   T_Dryer_4 : REAL ;
   T_air : REAL ;
   T_freon_Out_1 : REAL ;
   T_freon_Out_2 : REAL ;
   Dewpoint : REAL ;
  END_STRUCT ;	
BEGIN
END_DATA_BLOCK

DATA_BLOCK "PO2_AI2"	// DB 133
VERSION : 0.1
  STRUCT
   B_0 : BYTE ;
   B_1 : BYTE ;
   B_2 : BYTE ;
   B_3 : BYTE ;
  END_STRUCT ;	
BEGIN
END_DATA_BLOCK

DATA_BLOCK "DI_Bytes"	// DB 134
VERSION : 0.1
  STRUCT
   B_0 : BYTE ;
   B_1 : BYTE ;
   B_2 : BYTE ;
   B_3 : BYTE ;
   B_4 : BYTE ;
   B_5 : BYTE ;
   B_6 : BYTE ;
   B_7 : BYTE ;
   B_8 : BYTE ;
   B_9 : BYTE ;
   B_10 : BYTE ;
   B_11 : BYTE ;
   B_12 : BYTE ;
  END_STRUCT ;	
BEGIN
END_DATA_BLOCK

DATA_BLOCK "PCV10_PID_Vars"	// DB 135
VERSION : 0.1
  STRUCT
   rSetPressure : REAL ;
   rKp : REAL ;
   tKi : TIME  := T#3M20S;
   tKd : TIME ;
   rSetManualPercent : REAL ;
   xManualOn : BOOL ;
   rOut : REAL ;
  END_STRUCT ;	
BEGIN
   tKi := T#3M20S;
END_DATA_BLOCK

DATA_BLOCK "PCV21_PID_Vars"	// DB 136
VERSION : 0.1
  STRUCT
   rSetPressure : REAL ;
   rKp : REAL ;
   tKi : TIME  := T#3M20S;
   tKd : TIME ;
   rSetManualPercent : REAL ;
   xManualOn : BOOL ;
   rOut : REAL ;
  END_STRUCT ;	
BEGIN
   tKi := T#3M20S;
END_DATA_BLOCK

DATA_BLOCK "PCV22_PID_Vars"	// DB 137
VERSION : 0.1
  STRUCT
   rSetPressure : REAL ;
   rKp : REAL ;
   tKi : TIME  := T#3M20S;
   tKd : TIME ;
   rSetManualPercent : REAL ;
   xManualOn : BOOL ;
   rOut : REAL ;
  END_STRUCT ;	
BEGIN
   tKi := T#3M20S;
END_DATA_BLOCK

DATA_BLOCK "PCV25_PID_Vars"	// DB 138
VERSION : 0.1
  STRUCT
   rSetPressure : REAL ;
   rKp : REAL ;
   tKi : TIME  := T#3M20S;
   tKd : TIME ;
   rSetManualPercent : REAL ;
   xManualOn : BOOL ;
   rOut : REAL ;
  END_STRUCT ;	
BEGIN
   tKi := T#3M20S;
END_DATA_BLOCK

DATA_BLOCK "ValvesVars"	// DB 139
VERSION : 0.1
  STRUCT
   xCmdOpn_ZB1 : BOOL ;
   xCmdOpn_ZB2 : BOOL ;
   xCmdOpn_ZB3 : BOOL ;
   xCmdOpn_ZB4 : BOOL ;
   xCmdCls_ZB1 : BOOL ;
   xCmdCls_ZB2 : BOOL ;
   xCmdCls_ZB3 : BOOL ;
   xCmdCls_ZB4 : BOOL ;
   xCmdStop_ZB1 : BOOL ;
   xCmdStop_ZB2 : BOOL ;
   xCmdStop_ZB3 : BOOL ;
   xCmdStop_ZB4 : BOOL ;
   xCmdOpnManual_ZB1 : BOOL ;
   xCmdOpnManual_ZB2 : BOOL ;
   xCmdOpnManual_ZB3 : BOOL ;
   xCmdOpnManual_ZB4 : BOOL ;
   xCmdClsManual_ZB1 : BOOL ;
   xCmdClsManual_ZB2 : BOOL ;
   xCmdClsManual_ZB3 : BOOL ;
   xCmdClsManual_ZB4 : BOOL ;
   xCmdStopManual_ZB1 : BOOL ;
   xCmdStopManual_ZB2 : BOOL ;
   xCmdStopManual_ZB3 : BOOL ;
   xCmdStopManual_ZB4 : BOOL ;
   xManual_ZB1 : BOOL ;
   xManual_ZB2 : BOOL ;
   xManual_ZB3 : BOOL ;
   xManual_ZB4 : BOOL ;
   bAlm_ZB1 : BYTE ;
   bAlm_ZB2 : BYTE ;
   bAlm_ZB3 : BYTE ;
   bAlm_ZB4 : BYTE ;
  END_STRUCT ;	
BEGIN
END_DATA_BLOCK

DATA_BLOCK "SensorsAlarmSettings"	// DB 140
VERSION : 0.1
  STRUCT
   One_PIR7_Min : REAL  := 1.000000e+001;	//CompressedAirPressureAfter_KB_1_1
   One_PIR7_Max : REAL ;	//CompressedAirPressureAfter_KB_1_1
   Two_PIR7_Min : REAL ;	//CompressedAirPressureAfter_KB_1_2
   Two_PIR7_Max : REAL ;	//CompressedAirPressureAfter_KB_1_2
   One_PIR6_Min : REAL ;	//N_PressureAfter_KZA_1_1
   One_PIR6_Max : REAL ;	//N_PressureAfter_KZA_1_1
   Two_PIR6_Min : REAL ;	//N_PressureAfter_KZA_1_2
   Two_PIR6_Max : REAL ;	//N_PressureAfter_KZA_1_2
   PIR8_Min : REAL ;	//CompressedAirPressureAfter_KB_2
   PIR8_Max : REAL ;	//CompressedAirPressureAfter_KB_2
   Two_PIR20_Min : REAL ;	//N_PressureAfter_KZA_2_2
   Two_PIR20_Max : REAL ;	//N_PressureAfter_KZA_2_2
   TIR10_Min : REAL ;	//N_PressureIntoSystem
   TIR10_Max : REAL ;	//N_PressureIntoSystem
   FIR10_Min : REAL ;	//N_Consume
   FIR10_Max : REAL ;	//N_Consume
   PIR5_Min : REAL ;	//N_PressureIntoSystem
   PIR5_Max : REAL ;	//N_PressureIntoSystem
   FIR5_Min : REAL ;	//N_ConsumeSystem
   FIR5_Max : REAL ;	//N_ConsumeSystem
   PIRC21_Min : REAL ;	//N_PressureDiagn
   PIRC21_Max : REAL ;	//N_PressureDiagn
   One_PIR27_Min : REAL ;	//N_PressureAfter_PB_2_1
   One_PIR27_Max : REAL ;	//N_PressureAfter_PB_2_1
   QIRAH3_Min : REAL ;	//O2_Consis_KZA_1_1_2
   QIRAH3_Max : REAL ;	//O2_Consis_KZA_1_1_2
   Two_PIR27_Min : REAL ;	//AirPressure_PB_2_2
   Two_PIR27_Max : REAL ;	//AirPressure_PB_2_2
   PIR4_Min : REAL ;	//AirPressure
   PIR4_Max : REAL ;	//AirPressure
   FIR_4_Min : REAL ;	//CompressedAirConsum
   FIR_4_Max : REAL ;	//CompressedAirConsum
   PIRC22_Min : REAL ;	//AirPressure_PIRC22
   PIRC22_Max : REAL ;	//AirPressure_PIRC22
   PIRC23_Min : REAL ;	//AirPressure_PBT_1
   PIRC23_Max : REAL ;	//AirPressure_PBT_1
   PIRC24_Min : REAL ;	//AirPressure_PBK_1
   PIRC24_Max : REAL ;	//AirPressure_PBK_1
   PIRC25_Min : REAL ;	//AirPressure
   PIRC25_Max : REAL ;	//AirPressure
   FIR_25_Min : REAL ;	//CompressedAirConsum
   FIR_25_Max : REAL ;	//CompressedAirConsum
   One_PIRC26_Min : REAL ;	//AirPressure_PB_1_1
   One_PIRC26_Max : REAL ;	//AirPressure_PB_1_1
   Two_PIRC26_Min : REAL ;	//AirPressure_PB_1_2
   Two_PIRC26_Max : REAL ;	//AirPressure_PB_1_2
   PIRC_C10_Min : REAL ;	//N_Temp
   PIRC_C10_Max : REAL ;	//N_Temp
   TIR5_Min : REAL ;	//N_Temp
   TIR5_Max : REAL ;	//N_Temp
   TIR4_Min : REAL ;	//Air_Temp
   TIR4_Max : REAL ;	//Air_Temp
   TIR25_Min : REAL ;	//Air_Temp
   TIR25_Max : REAL ;	//Air_Temp
   AIR1_Min : REAL ;	//Air_Wetness_AIR1
   AIR1_Max : REAL ;	//Air_Wetness_AIR1
   One_PIR20_Min : REAL ;	//N_PressureAfter_KZA_2_2
   One_PIR20_Max : REAL ;	//N_PressureAfter_KZA_2_2
   QIRAH4H4_Min : REAL ;
   QIRAH4H4_Max : REAL ;
  END_STRUCT ;	
BEGIN
   One_PIR7_Min := 1.000000e+01;
END_DATA_BLOCK

DATA_BLOCK "BD_MaxMin"	// DB 141
VERSION : 0.1
  STRUCT
   PressureVesselA_Min : REAL ;
   PressureVesselB_Min : REAL ;
   InletDryer_Min : REAL ;
   HeaterOut_Min : REAL ;
   RegenerAirOutlet_Min : REAL ;
   DryerPresDewpoint_Min : REAL ;
   PressureVesselA_Max : REAL ;
   PressureVesselB_Max : REAL ;
   InletDryer_Max : REAL ;
   HeaterOut_Max : REAL ;
   RegenerAirOutlet_Max : REAL ;
   DryerPresDewpoint_Max : REAL ;
  END_STRUCT ;	
BEGIN
END_DATA_BLOCK

DATA_BLOCK "GA1_1_MinMax"	// DB 142
VERSION : 0.1
  STRUCT
   AirGeneratorIn_Min : REAL ;
   PressureVesselA_Min : REAL ;
   PressureVesselB_Min : REAL ;
   NitrogenOutlet_Min : REAL ;
   AirGeneratorIn1_Min : REAL ;
   DryerPressDewpoint_Min : REAL ;
   NitrogenDewpoint_Min : REAL ;
   OutletFlow_Min : REAL ;
   OxygenPurity_Min : REAL ;
   AirGeneratorIn_Max : REAL ;
   PressureVesselA_Max : REAL ;
   PressureVesselB_Max : REAL ;
   NitrogenOutlet_Max : REAL ;
   AirGeneratorIn1_Max : REAL ;
   DryerPressDewpoint_Max : REAL ;
   NitrogenDewpoint_Max : REAL ;
   OutletFlow_Max : REAL ;
   OxygenPurity_Max : REAL ;
  END_STRUCT ;	
BEGIN
END_DATA_BLOCK

DATA_BLOCK "GA1_2_MinMax"	// DB 143
VERSION : 0.1
  STRUCT
   AirGeneratorIn_Min : REAL ;
   PressureVesselA_Min : REAL ;
   PressureVesselB_Min : REAL ;
   NitrogenOutlet_Min : REAL ;
   AirGeneratorIn1_Min : REAL ;
   DryerPressDewpoint_Min : REAL ;
   NitrogenDewpoint_Min : REAL ;
   OutletFlow_Min : REAL ;
   OxygenPurity_Min : REAL ;
   AirGeneratorIn_Max : REAL ;
   PressureVesselA_Max : REAL ;
   PressureVesselB_Max : REAL ;
   NitrogenOutlet_Max : REAL ;
   AirGeneratorIn1_Max : REAL ;
   DryerPressDewpoint_Max : REAL ;
   NitrogenDewpoint_Max : REAL ;
   OutletFlow_Max : REAL ;
   OxygenPurity_Max : REAL ;
  END_STRUCT ;	
BEGIN
END_DATA_BLOCK

DATA_BLOCK "GA2_1_MinMax"	// DB 144
VERSION : 0.1
  STRUCT
   AirGeneratorIn_Min : REAL ;
   PressureVesselA_Min : REAL ;
   PressureVesselB_Min : REAL ;
   NitrogenOutlet_Min : REAL ;
   AirGeneratorIn1_Min : REAL ;
   DryerPressDewpoint_Min : REAL ;
   NitrogenDewpoint_Min : REAL ;
   OutletFlow_Min : REAL ;
   OxygenPurity_Min : REAL ;
   AirGeneratorIn_Max : REAL ;
   PressureVesselA_Max : REAL ;
   PressureVesselB_Max : REAL ;
   NitrogenOutlet_Max : REAL ;
   AirGeneratorIn1_Max : REAL ;
   DryerPressDewpoint_Max : REAL ;
   NitrogenDewpoint_Max : REAL ;
   OutletFlow_Max : REAL ;
   OxygenPurity_Max : REAL ;
  END_STRUCT ;	
BEGIN
END_DATA_BLOCK

DATA_BLOCK "GA2_2_MinMax"	// DB 145
VERSION : 0.1
  STRUCT
   AirGeneratorIn_Min : REAL ;
   PressureVesselA_Min : REAL ;
   PressureVesselB_Min : REAL ;
   NitrogenOutlet_Min : REAL ;
   AirGeneratorIn1_Min : REAL ;
   DryerPressDewpoint_Min : REAL ;
   NitrogenDewpoint_Min : REAL ;
   OutletFlow_Min : REAL ;
   OxygenPurity_Min : REAL ;
   AirGeneratorIn_Max : REAL ;
   PressureVesselA_Max : REAL ;
   PressureVesselB_Max : REAL ;
   NitrogenOutlet_Max : REAL ;
   AirGeneratorIn1_Max : REAL ;
   DryerPressDewpoint_Max : REAL ;
   NitrogenDewpoint_Max : REAL ;
   OutletFlow_Max : REAL ;
   OxygenPurity_Max : REAL ;
  END_STRUCT ;	
BEGIN
END_DATA_BLOCK

DATA_BLOCK "KB1_1_MinMax"	// DB 146
VERSION : 0.1
  STRUCT
   InputPressure_Min : REAL ;
   PressChngOnFiltr_Min : REAL ;
   OilPressure_Min : REAL ;
   PromCoolerPres_Min : REAL ;
   TafterCompressor_Min : REAL ;
   TafterStep_1_Min : REAL ;
   TafterStep_2_Min : REAL ;
   TafterStep_3_Min : REAL ;
   TinputCoolWater_Min : REAL ;
   TwaterAfterStepND_Min : REAL ;
   ToutCoolWater_Min : REAL ;
   Toil_Min : REAL ;
   Tmotor_U1_Min : REAL ;
   Tmotor_V1_Min : REAL ;
   Tmotor_W1_Min : REAL ;
   InputPressure_Max : REAL ;
   PressChngOnFiltr_Max : REAL ;
   OilPressure_Max : REAL ;
   PromCoolerPres_Max : REAL ;
   TafterCompressor_Max : REAL ;
   TafterStep_1_Max : REAL ;
   TafterStep_2_Max : REAL ;
   TafterStep_3_Max : REAL ;
   TinputCoolWater_Max : REAL ;
   TwaterAfterStepND_Max : REAL ;
   ToutCoolWater_Max : REAL ;
   Toil_Max : REAL ;
   Tmotor_U1_Max : REAL ;
   Tmotor_V1_Max : REAL ;
   Tmotor_W1_Max : REAL ;
  END_STRUCT ;	
BEGIN
END_DATA_BLOCK

DATA_BLOCK "KB1_2_MinMax"	// DB 147
VERSION : 0.1
  STRUCT
   InputPressure_Min : REAL ;
   PressChngOnFiltr_Min : REAL ;
   OilPressure_Min : REAL ;
   PromCoolerPres_Min : REAL ;
   TafterCompressor_Min : REAL ;
   TafterStep_1_Min : REAL ;
   TafterStep_2_Min : REAL ;
   TafterStep_3_Min : REAL ;
   TinputCoolWater_Min : REAL ;
   TwaterAfterStepND_Min : REAL ;
   ToutCoolWater_Min : REAL ;
   Toil_Min : REAL ;
   Tmotor_U1_Min : REAL ;
   Tmotor_V1_Min : REAL ;
   Tmotor_W1_Min : REAL ;
   InputPressure_Max : REAL ;
   PressChngOnFiltr_Max : REAL ;
   OilPressure_Max : REAL ;
   PromCoolerPres_Max : REAL ;
   TafterCompressor_Max : REAL ;
   TafterStep_1_Max : REAL ;
   TafterStep_2_Max : REAL ;
   TafterStep_3_Max : REAL ;
   TinputCoolWater_Max : REAL ;
   TwaterAfterStepND_Max : REAL ;
   ToutCoolWater_Max : REAL ;
   Toil_Max : REAL ;
   Tmotor_U1_Max : REAL ;
   Tmotor_V1_Max : REAL ;
   Tmotor_W1_Max : REAL ;
  END_STRUCT ;	
BEGIN
END_DATA_BLOCK

DATA_BLOCK "KD2_ManMax"	// DB 148
VERSION : 0.1
  STRUCT
   OilPressureReductor_Min : REAL ;
   PressChangeOnFiltr_Min : REAL ;
   PressChngeOnOilFiltr_Min : REAL ;
   Step3OutPressure_Min : REAL ;
   ToilReductor_Min : REAL ;
   TinputCoolWater_Min : REAL ;
   TinputStep_2_Min : REAL ;
   TinputStep_3_Min : REAL ;
   TafterCompressor_Min : REAL ;
   ToilTank_Min : REAL ;
   Tmotor_U1_Min : REAL ;
   Tmotor_V1_Min : REAL ;
   Tmotor_W1_Min : REAL ;
   OutPressure_Min : REAL ;
   Aject2Step_Min : REAL ;
   PchangeStep2_Min : REAL ;
   TmotorBearier_D_End_Min : REAL ;
   TmotorBearier_ND_End_Min : REAL ;
   Vibration_1_Min : REAL ;
   Vibration_2_Min : REAL ;
   Vibration_3_Min : REAL ;
   OilPressureReductor_Max : REAL ;
   PressChangeOnFiltr_Max : REAL ;
   PressChngeOnOilFiltr_Max : REAL ;
   Step3OutPressure_Max : REAL ;
   ToilReductor_Max : REAL ;
   TinputCoolWater_Max : REAL ;
   TinputStep_2_Max : REAL ;
   TinputStep_3_Max : REAL ;
   TafterCompressor_Max : REAL ;
   ToilTank_Max : REAL ;
   Tmotor_U1_Max : REAL ;
   Tmotor_V1_Max : REAL ;
   Tmotor_W1_Max : REAL ;
   OutPressure_Max : REAL ;
   Aject2Step_Max : REAL ;
   PchangeStep2_Max : REAL ;
   TmotorBearier_D_End_Max : REAL ;
   TmotorBearier_ND_End_Max : REAL ;
   Vibration_1_Max : REAL ;
   Vibration_2_Max : REAL ;
   Vibration_3_Max : REAL ;
  END_STRUCT ;	
BEGIN
END_DATA_BLOCK

DATA_BLOCK "PO1_1_MaxMin"	// DB 149
VERSION : 0.1
  STRUCT
   CondPressure_Min : REAL ;
   EvapPressureComp_Min : REAL ;
   EvapPressHE_1_Min : REAL ;
   EvapPressHE_2_Min : REAL ;
   Dewpoint_1_Min : REAL ;
   Freon_1_Min : REAL ;
   Dewpoint_2_Min : REAL ;
   Freon_11_Min : REAL ;
   ToutAir_Min : REAL ;
   TfreonIn_Min : REAL ;
   TfreonOut_Min : REAL ;
   CondPressure_Max : REAL ;
   EvapPressureComp_Max : REAL ;
   EvapPressHE_1_Max : REAL ;
   EvapPressHE_2_Max : REAL ;
   Dewpoint_1_Max : REAL ;
   Freon_1_Max : REAL ;
   Dewpoint_2_Max : REAL ;
   Freon_11_Max : REAL ;
   ToutAir_Max : REAL ;
   TfreonIn_Max : REAL ;
   TfreonOut_Max : REAL ;
  END_STRUCT ;	
BEGIN
END_DATA_BLOCK

DATA_BLOCK "PO1_2_MinMax"	// DB 150
VERSION : 0.1
  STRUCT
   CondPressure_Min : REAL ;
   EvapPressureComp_Min : REAL ;
   EvapPressHE_1_Min : REAL ;
   EvapPressHE_2_Min : REAL ;
   Dewpoint_1_Min : REAL ;
   Freon_1_Min : REAL ;
   Dewpoint_2_Min : REAL ;
   Freon_11_Min : REAL ;
   ToutAir_Min : REAL ;
   TfreonIn_Min : REAL ;
   TfreonOut_Min : REAL ;
   CondPressure_Max : REAL ;
   EvapPressureComp_Max : REAL ;
   EvapPressHE_1_Max : REAL ;
   EvapPressHE_2_Max : REAL ;
   Dewpoint_1_Max : REAL ;
   Freon_1_Max : REAL ;
   Dewpoint_2_Max : REAL ;
   Freon_11_Max : REAL ;
   ToutAir_Max : REAL ;
   TfreonIn_Max : REAL ;
   TfreonOut_Max : REAL ;
  END_STRUCT ;	
BEGIN
END_DATA_BLOCK

DATA_BLOCK "ProcessSettings"	// DB 151
VERSION : 0.1
  STRUCT
   tKB1StartDelay : S5TIME  := S5T#10M;	//Temporary placeholder variable
   tKB2tartDelay : S5TIME  := S5T#10M10S;
   rPressureSet_1 : REAL  := 8.500000e+000;
   rPressureSet_2 : REAL  := 8.500000e+000;
  END_STRUCT ;	
BEGIN
   tKB1StartDelay := S5T#10M;
   tKB2tartDelay := S5T#10M10S;
   rPressureSet_1 := 8.500000e+00;
   rPressureSet_2 := 8.500000e+00;
END_DATA_BLOCK

DATA_BLOCK "ProcessVars"	// DB 152
VERSION : 0.1
  STRUCT
   xStartProc1 : BOOL ;	//Temporary placeholder variable
   xStartProc2 : BOOL ;	//Temporary placeholder variable
  END_STRUCT ;	
BEGIN
END_DATA_BLOCK

DATA_BLOCK "PrepareStartStop"	// DB 153
VERSION : 0.1
  STRUCT
   xBD_Start : BOOL ;
   xBD_Stop : BOOL ;
   xKB1_1_Start : BOOL ;
   xKB1_1_Stop : BOOL ;
   xKB1_2_Start : BOOL ;
   xKB1_2_Stop : BOOL ;
   xKB2_Start : BOOL ;
   xKB2_Stop : BOOL ;
   xPO1_1_Start : BOOL ;
   xPO1_1_Stop : BOOL ;
   xPO1_2_Start : BOOL ;
   xPO1_2_Stop : BOOL ;
   xGA1_1_Start : BOOL ;
   xGA1_1_Stop : BOOL ;
   xGA1_2_Start : BOOL ;
   xGA1_2_Stop : BOOL ;
   xGA2_1_Start : BOOL ;
   xGA2_1_Stop : BOOL ;
   xGA2_2_Start : BOOL ;
   xGA2_2_Stop : BOOL ;
   xKD_Start : BOOL ;
   xKD_Stop : BOOL ;
   xPO2_Start : BOOL ;
   xPO2_Stop : BOOL ;
  END_STRUCT ;	
BEGIN
END_DATA_BLOCK

DATA_BLOCK "PO2_Coils"	// DB 154
VERSION : 0.1
  STRUCT
   B_0 : BYTE ;
   B_1 : BYTE ;
   Running_Stopped : BOOL  := TRUE;
   Load_Unload : BOOL ;
   General_Warning : BOOL ;
   GeneralShutdownWarning : BOOL ;
   GeneralShutdown : BOOL ;
   GeneralService : BOOL ;
   GeneralStartFailure : BOOL ;
   EmergencyStop : BOOL ;
   Automatic_Manual : BOOL ;
   Remote_Local : BOOL ;
  END_STRUCT ;	
BEGIN
END_DATA_BLOCK

DATA_BLOCK "PO2_MinMax"	// DB 155
VERSION : 0.1
  STRUCT
   T_Dryer_1_Min : REAL ;
   T_Dryer_2_Min : REAL ;
   T_Dryer_3_Min : REAL ;
   T_Dryer_4_Min : REAL ;
   T_air_Min : REAL ;
   T_freon_Out_1_Min : REAL ;
   T_freon_Out_2_Min : REAL ;
   Dewpoint_Min : REAL ;
   T_Dryer_1_Max : REAL ;
   T_Dryer_2_Max : REAL ;
   T_Dryer_3_Max : REAL ;
   T_Dryer_4_Max : REAL ;
   T_air_Max : REAL ;
   T_freon_Out_1_Max : REAL ;
   T_freon_Out_2_Max : REAL ;
   Dewpoint_Max : REAL ;
  END_STRUCT ;	
BEGIN
END_DATA_BLOCK

DATA_BLOCK DB 200
AUTHOR : T.HAJNAL
FAMILY : MODBUS
VERSION : 0.0
"MBMAREQ"
BEGIN
END_DATA_BLOCK

DATA_BLOCK DB 201
AUTHOR : T.HAJNAL
FAMILY : MODBUS
VERSION : 0.0
"MBMAREQ"
BEGIN
END_DATA_BLOCK

DATA_BLOCK DB 202
AUTHOR : T.HAJNAL
FAMILY : MODBUS
VERSION : 0.0
"MBMAREQ"
BEGIN
END_DATA_BLOCK

DATA_BLOCK DB 203
AUTHOR : T.HAJNAL
FAMILY : MODBUS
VERSION : 0.0
"MBMAREQ"
BEGIN
END_DATA_BLOCK

DATA_BLOCK DB 204
AUTHOR : T.HAJNAL
FAMILY : MODBUS
VERSION : 0.0
"MBMAREQ"
BEGIN
END_DATA_BLOCK

DATA_BLOCK DB 205
AUTHOR : T.HAJNAL
FAMILY : MODBUS
VERSION : 0.0
"MBMAREQ"
BEGIN
END_DATA_BLOCK

DATA_BLOCK DB 206
AUTHOR : T.HAJNAL
FAMILY : MODBUS
VERSION : 0.0
"MBMAREQ"
BEGIN
END_DATA_BLOCK

DATA_BLOCK DB 207
AUTHOR : T.HAJNAL
FAMILY : MODBUS
VERSION : 0.0
"MBMAREQ"
BEGIN
END_DATA_BLOCK

DATA_BLOCK DB 208
AUTHOR : T.HAJNAL
FAMILY : MODBUS
VERSION : 0.0
"MBMAREQ"
BEGIN
END_DATA_BLOCK

DATA_BLOCK DB 209
AUTHOR : T.HAJNAL
FAMILY : MODBUS
VERSION : 0.0
"MBMAREQ"
BEGIN
END_DATA_BLOCK

DATA_BLOCK DB 210
AUTHOR : T.HAJNAL
FAMILY : MODBUS
VERSION : 0.0
"MBMAREQ"
BEGIN
END_DATA_BLOCK

DATA_BLOCK DB 211
AUTHOR : T.HAJNAL
FAMILY : MODBUS
VERSION : 0.0
"MBMAREQ"
BEGIN
END_DATA_BLOCK

DATA_BLOCK DB 330
VERSION : 0.0
"Valve_PID"
BEGIN
END_DATA_BLOCK

DATA_BLOCK DB 331
VERSION : 0.0
"Valve_PID"
BEGIN
END_DATA_BLOCK

DATA_BLOCK DB 332
VERSION : 0.0
"Valve_PID"
BEGIN
END_DATA_BLOCK

DATA_BLOCK DB 333
VERSION : 0.0
"Valve_PID"
BEGIN
END_DATA_BLOCK

DATA_BLOCK DB 500
VERSION : 0.0
"BD_GetReals"
BEGIN
END_DATA_BLOCK

DATA_BLOCK DB 501
VERSION : 0.0
"KB1_1_GetReals"
BEGIN
END_DATA_BLOCK

DATA_BLOCK DB 502
VERSION : 0.0
"KB1_2_GetReals"
BEGIN
END_DATA_BLOCK

DATA_BLOCK DB 503
VERSION : 0.0
"KB2_GetReals"
BEGIN
END_DATA_BLOCK

DATA_BLOCK DB 504
VERSION : 0.0
"PO1_1_GetReals"
BEGIN
END_DATA_BLOCK

DATA_BLOCK DB 505
VERSION : 0.0
"PO1_2_GetReals"
BEGIN
END_DATA_BLOCK

DATA_BLOCK DB 506
VERSION : 0.0
"GA1_1_GetReal"
BEGIN
END_DATA_BLOCK

DATA_BLOCK DB 507
VERSION : 0.0
"GA1_2_GetReals"
BEGIN
END_DATA_BLOCK

DATA_BLOCK DB 508
VERSION : 0.0
"GA2_1_GetReals"
BEGIN
END_DATA_BLOCK

DATA_BLOCK DB 509
VERSION : 0.0
"GA2_2_GetReals"
BEGIN
END_DATA_BLOCK

DATA_BLOCK DB 510
VERSION : 0.0
"KD_GetReals"
BEGIN
END_DATA_BLOCK

DATA_BLOCK DB 511
VERSION : 0.0
"BD_GetOutputs"
BEGIN
END_DATA_BLOCK

DATA_BLOCK DB 512
VERSION : 0.0
"PO1_1_GetOutputs"
BEGIN
END_DATA_BLOCK

DATA_BLOCK DB 513
VERSION : 0.0
"PO1_2_GetOutputs"
BEGIN
END_DATA_BLOCK

DATA_BLOCK DB 514
VERSION : 0.0
"GA1_1_GetOutputs"
BEGIN
END_DATA_BLOCK

DATA_BLOCK DB 515
VERSION : 0.0
"GA1_2_GetOutputs"
BEGIN
END_DATA_BLOCK

DATA_BLOCK DB 516
VERSION : 0.0
"GA2_1_GetOutputs"
BEGIN
END_DATA_BLOCK

DATA_BLOCK DB 517
VERSION : 0.0
"GA2_2_GetOutputs"
BEGIN
END_DATA_BLOCK

DATA_BLOCK DB 518
VERSION : 0.0
"GetStartStopBytes"
BEGIN
END_DATA_BLOCK

DATA_BLOCK DB 519
VERSION : 0.0
"PO2_GetReals"
BEGIN
END_DATA_BLOCK

DATA_BLOCK DB 700
VERSION : 0.0
"ModbusCoils"
BEGIN
END_DATA_BLOCK

DATA_BLOCK DB 701
VERSION : 0.0
"ModbusReal"
BEGIN
END_DATA_BLOCK

DATA_BLOCK DB 702
VERSION : 0.0
"ModbusOutputs"
BEGIN
END_DATA_BLOCK

DATA_BLOCK DB 703
VERSION : 0.0
"ModbusStartStop"
BEGIN
END_DATA_BLOCK

DATA_BLOCK "ZB1"	// DB 777
VERSION : 0.0
"DO_Valve"
BEGIN
END_DATA_BLOCK

DATA_BLOCK "ZB2"	// DB 778
VERSION : 0.0
"DO_Valve"
BEGIN
END_DATA_BLOCK

DATA_BLOCK "ZB3"	// DB 779
VERSION : 0.0
"DO_Valve"
BEGIN
END_DATA_BLOCK

DATA_BLOCK "ZB4"	// DB 780
VERSION : 0.0
"DO_Valve"
BEGIN
END_DATA_BLOCK

DATA_BLOCK "ValvesPrgDB"	// DB 781
VERSION : 0.0
"ValvesPrg"
BEGIN
END_DATA_BLOCK

DATA_BLOCK DB 782
VERSION : 0.0
"ValvesPrg"
BEGIN
END_DATA_BLOCK

DATA_BLOCK DB 791
VERSION : 0.0
"Valve_PID"
BEGIN
END_DATA_BLOCK

DATA_BLOCK DB 792
VERSION : 0.0
"Valve_PID"
BEGIN
END_DATA_BLOCK

DATA_BLOCK DB 793
VERSION : 0.0
"Valve_PID"
BEGIN
END_DATA_BLOCK

DATA_BLOCK DB 794
VERSION : 0.0
"Valve_PID"
BEGIN
END_DATA_BLOCK

DATA_BLOCK DB 800
VERSION : 0.0
"GetAll"
BEGIN
END_DATA_BLOCK

DATA_BLOCK DB 801
VERSION : 0.0
"ModbusAll"
BEGIN
END_DATA_BLOCK

DATA_BLOCK DB 802
AUTHOR : T.HAJNAL
FAMILY : MODBUS
VERSION : 0.0
"MBMA341"
BEGIN
END_DATA_BLOCK

DATA_BLOCK DB 901
AUTHOR : T.HAJNAL
FAMILY : MODBUS
VERSION : 0.0
"MBMAREQ"
BEGIN
END_DATA_BLOCK

DATA_BLOCK DB 902
AUTHOR : T.HAJNAL
FAMILY : MODBUS
VERSION : 0.0
"MBMAREQ"
BEGIN
END_DATA_BLOCK

DATA_BLOCK DB 903
AUTHOR : T.HAJNAL
FAMILY : MODBUS
VERSION : 0.0
"MBMAREQ"
BEGIN
END_DATA_BLOCK

DATA_BLOCK DB 904
AUTHOR : T.HAJNAL
FAMILY : MODBUS
VERSION : 0.0
"MBMAREQ"
BEGIN
END_DATA_BLOCK

DATA_BLOCK DB 1000
VERSION : 0.0
"InToVars"
BEGIN
END_DATA_BLOCK

DATA_BLOCK DB 1001
VERSION : 0.0
"ModbusAll"
BEGIN
END_DATA_BLOCK

DATA_BLOCK DB 1002
AUTHOR : T.HAJNAL
FAMILY : MODBUS
VERSION : 0.0
"MBMA341"
BEGIN
END_DATA_BLOCK

DATA_BLOCK DB 1003
VERSION : 0.0
"prProcess"
BEGIN
END_DATA_BLOCK

DATA_BLOCK DB 1004
VERSION : 0.0
"prDevices"
BEGIN
END_DATA_BLOCK

DATA_BLOCK DB 1010
VERSION : 0.0
"InToVarsST"
BEGIN
END_DATA_BLOCK

DATA_BLOCK DB 1011
VERSION : 0.0
"DI_ToVars"
BEGIN
END_DATA_BLOCK

DATA_BLOCK DB 1110
AUTHOR : SIMATIC
FAMILY : ICONT
VERSION : 0.0
"CONT_C"
BEGIN
END_DATA_BLOCK

DATA_BLOCK DB 1111
AUTHOR : T.HAJNAL
FAMILY : MODBUS
VERSION : 0.0
"MBMAREQ"
BEGIN
END_DATA_BLOCK

DATA_BLOCK DB 1500
VERSION : 0.0
"fbImpulsValveSCL"
BEGIN
END_DATA_BLOCK

DATA_BLOCK DB 1501
VERSION : 0.0
"fbImpulsValveSCL"
BEGIN
END_DATA_BLOCK

DATA_BLOCK DB 1502
VERSION : 0.0
"fbImpulsValveSCL"
BEGIN
END_DATA_BLOCK

DATA_BLOCK DB 1503
VERSION : 0.0
"fbImpulsValveSCL"
BEGIN
END_DATA_BLOCK

DATA_BLOCK DB 2000
VERSION : 0.0
"fbProcess_1"
BEGIN
END_DATA_BLOCK

DATA_BLOCK DB 2001
VERSION : 0.0
"fbProcess_1"
BEGIN
END_DATA_BLOCK

DATA_BLOCK DB 2100
VERSION : 0.0
"fbPO"
BEGIN
END_DATA_BLOCK

DATA_BLOCK DB 2101
VERSION : 0.0
"fbPO"
BEGIN
END_DATA_BLOCK

DATA_BLOCK DB 2102
VERSION : 0.0
"fbPO"
BEGIN
END_DATA_BLOCK

DATA_BLOCK DB 2103
VERSION : 0.0
"fbKB"
BEGIN
END_DATA_BLOCK

DATA_BLOCK DB 2104
VERSION : 0.0
"fbKB"
BEGIN
END_DATA_BLOCK

DATA_BLOCK DB 2105
VERSION : 0.0
"fbKB"
BEGIN
END_DATA_BLOCK

DATA_BLOCK DB 2106
VERSION : 0.0
"fbKZA"
BEGIN
END_DATA_BLOCK

DATA_BLOCK DB 2107
VERSION : 0.0
"fbKZA"
BEGIN
END_DATA_BLOCK

DATA_BLOCK DB 2108
VERSION : 0.0
"fbKZA"
BEGIN
END_DATA_BLOCK

DATA_BLOCK DB 2109
VERSION : 0.0
"fbKZA"
BEGIN
END_DATA_BLOCK

ORGANIZATION_BLOCK OB 1
TITLE = "Main Program Sweep (Cycle)"
VERSION : 0.1
VAR_TEMP
  OB1_EV_CLASS : BYTE ;	//Bits 0-3 = 1 (Coming event), Bits 4-7 = 1 (Event class 1)
  OB1_SCAN_1 : BYTE ;	//1 (Cold restart scan 1 of OB 1), 3 (Scan 2-n of OB 1)
  OB1_PRIORITY : BYTE ;	//Priority of OB Execution
  OB1_OB_NUMBR : BYTE ;	//1 (Organization block 1, OB1)
  OB1_RESERVED_1 : BYTE ;	//Reserved for system
  OB1_RESERVED_2 : BYTE ;	//Reserved for system
  OB1_PREV_CYCLE : INT ;	//Cycle time of previous OB1 scan (milliseconds)
  OB1_MIN_CYCLE : INT ;	//Minimum cycle time of OB1 (milliseconds)
  OB1_MAX_CYCLE : INT ;	//Maximum cycle time of OB1 (milliseconds)
  OB1_DATE_TIME : DATE_AND_TIME ;	//Date and time OB1 started
END_VAR
BEGIN
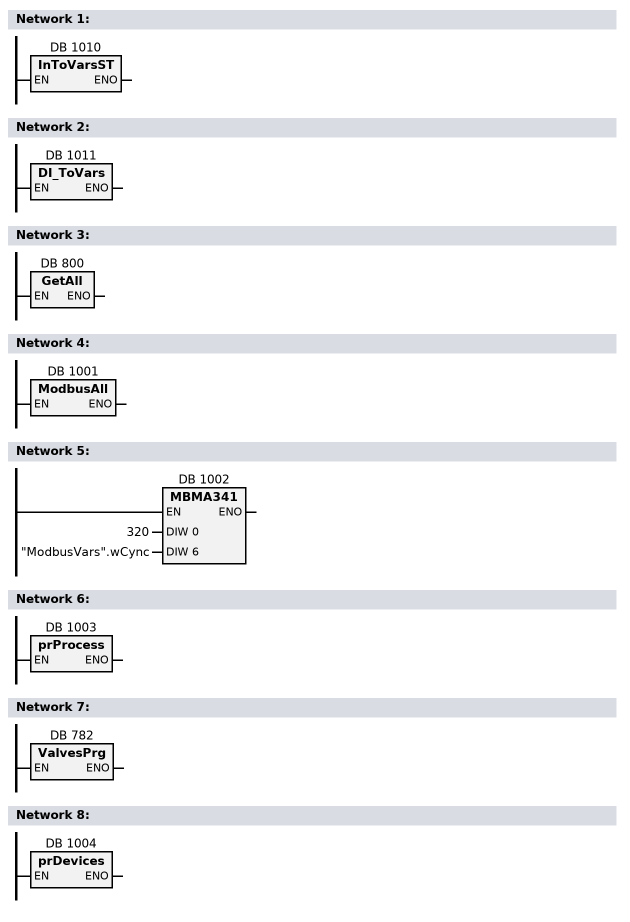
NETWORK
TITLE =
      CALL  "InToVarsST" , DB 1010;
      NOP   0;
NETWORK
TITLE =
      CALL  "DI_ToVars" , DB 1011;
      NOP   0;
NETWORK
TITLE =
      CALL  "GetAll" , DB 800;
      NOP   0;
NETWORK
TITLE =
      CALL  "ModbusAll" , DB 1001;
      NOP   0;
NETWORK
TITLE =
      CALL  "MBMA341" , DB 1002 (
           DIW 0                    := 320,
           DIW 6                    := "ModbusVars".wCync);
      NOP   0;
NETWORK
TITLE =
      CALL  "prProcess" , DB 1003;
      NOP   0;
NETWORK
TITLE =
      CALL  "ValvesPrg" , DB 782;
      NOP   0;
NETWORK
TITLE =
      CALL  "prDevices" , DB 1004;
      NOP   0;
END_ORGANIZATION_BLOCK

